(* CODESYS project StorageStation_CECCPrg.project

Project tree, tasks and I/O mapping:
  Device : CECC-D, Festo AG & Co. KG, order no. 574415, version 3.5.4.0
    application Application
      libraries: Standard, * (System); Festo_EXCM_3, 3.5.4.24 (Festo AG & Co. KG); Festo_CVE_3, 3.5.2.11 (Festo AG & Co. KG); VisuDialogs, * (System); CAA CiA 405, 3.5.3.0 (CAA Technical Workgroup)
      task MainTask (cyclic, interval t#20ms, priority 20) calls PLC_PRG
      task VISU_TASK (cyclic, interval 100 ms, priority 30) calls VisuElems.Visu_Prg
      program PLC_PRG [LD]
      global variables Globals
      image pool ImagePool
      global variables Store_Vars
      Visu/
        visualisation Storage_Scheme_new
        visualisation Optionen
        visualisation StorageVisu
        visualisation H_Portal
        visualisation Z_Axis
        visualisation generalControls
      Texts/
        text list Glob_TextList
        text list ARR_ZPOS
        text list ARR_XYPOS
        text list ARR_SPEED
        text list ARR_COLORCHOOSE
      PRGS/
        program prg_hlp [ST]
        program prg_connectCMMO [ST]
        program prg_DriveZAxis [ST]
        program prg_GlobalRef [ST]
        program prg_HomeEXCM [SFC]: Init_active
        program prg_RUNT [ST]
        program prg_HomeZAxis [SFC]
        program prg_startup [ST]
      Driver/
        program prg_DRIVER_CMMO [ST]
        program prg_CALL_DRIVES [FBD]
      EXCM/
        function block EXCM_CCON_CCPOS [ST]
        program EXCM_MANUALJOGG [FBD]
        program EXCM_POSCALC [ST]
        function block EXCM_SCON [ST]
        function block EXCM_SPOS [ST]
      global variables EXCM_Variables
      global variables IN_OUT_VARS
      FB/
        function block FB_Joggin [ST]
        function block FB_DriveZAxis [ST]
        function block FB_Store [ST]
        function block FB_Recognize [ST]
        function block FB_CalcRackPos [ST]
        function block FB_StoreSearch [ST]
        function block FB_DriveHPortal [ST]
        function block FB_SetStorePlace [ST]
        function block FB_Unstore [ST]
        function block FB_ClearStorePlace [ST]
    Onboard : CECC 14I/8O, Festo AG & Co. KG, order no. 
      , version 3.4.5.5
        unmapped channels: Onboard Input, Onboard Output
      Digital Inputs
          unmapped channels: Onboard Input
      Digital Outputs
          output qxGrab : BOOL  // Onboard Output.Byte0.Bit4
          unmapped channels: Onboard Output
    CANbus : CANbus, 3S - Smart Software Solutions GmbH, version 3.5.12.0
        settings: Baudrate = 1000 kbit/s
      CANopen_Manager : CANopen_Manager, 3S - Smart Software Solutions GmbH, version 3.5.10.0
          settings: Sync CycleTime in Microseconds = 8000; Synchronous Window Length = 0; Enable Heartbeat generation = FALSE; ConfigVersion = 50659584
        EXCM_2ST_C3_1 : EXCM-2ST-C3-1, Festo AG & Co. KG, order no. EXCM-CO, version Revision=16#00010000, FileVersion=2.1
            settings: NODEIDSAVED = 1; SDO Timeout = 1000000; EXPERTSETTINGS = TRUE; PDO 16#1400.COBID = 16#0201; PDO 16#1800.COBID = 16#0181; CCON_CPOS.Subindex = 16#00; REC_NR/VELOCITY.Subindex = 16#00; TARGET_POSX.Subindex = 16#00; TARGET_POSY.Subindex = 16#00; SCON_SPOS.Subindex = 16#00; ERROR_NR.Subindex = 16#00; ACT_POSX.Subindex = 16#00; ACT_POSY.Subindex = 16#00; SDO List.Set Guardtime.Index = 16#100C; SDO List.Set Guardtime.Subindex = 16#00; SDO List.Set Guardtime.Value = 16#00000000; SDO List.Set Guardtime.Size = 16; SDO List.Set Guardtime.AbortIfError = FALSE; SDO List.Set Guardtime.JumpToLine = FALSE; SDO List.Set Guardtime.Line = 0; SDO List.Set Lifetime.Index = 16#100D; SDO List.Set Lifetime.Subindex = 16#00; SDO List.Set Lifetime.Value = 16#00000000; SDO List.Set Lifetime.Size = 8; SDO List.Set Lifetime.AbortIfError = FALSE; SDO List.Set Lifetime.JumpToLine = FALSE; SDO List.Set Lifetime.Line = 0; SDO List.Disable Emcy CobID.Index = 16#1014; SDO List.Disable Emcy CobID.Subindex = 16#00; SDO List.Disable Emcy CobID.Value = 16#80000081; SDO List.Disable Emcy CobID.Size = 32; SDO List.Disable Emcy CobID.AbortIfError = FALSE; SDO List.Disable Emcy CobID.JumpToLine = FALSE; SDO List.Disable Emcy CobID.Line = 0; SDO List.Set Emcy CobID.Index = 16#1014; SDO List.Set Emcy CobID.Subindex = 16#00; SDO List.Set Emcy CobID.Value = 16#00000081; SDO List.Set Emcy CobID.Size = 32; SDO List.Set Emcy CobID.AbortIfError = FALSE; SDO List.Set Emcy CobID.JumpToLine = FALSE;
              SDO List.Set Emcy CobID.Line = 0; SDO List.Disable PDO.Index = 16#1400; SDO List.Disable PDO.Subindex = 16#01; SDO List.Disable PDO.Value = 16#80000201; SDO List.Disable PDO.Size = 32; SDO List.Disable PDO.AbortIfError = FALSE; SDO List.Disable PDO.JumpToLine = FALSE; SDO List.Disable PDO.Line = 0; SDO List.Set transmission type.Index = 16#1400; SDO List.Set transmission type.Subindex = 16#02; SDO List.Set transmission type.Value = 16#FF; SDO List.Set transmission type.Size = 8; SDO List.Set transmission type.AbortIfError = FALSE; SDO List.Set transmission type.JumpToLine = FALSE; SDO List.Set transmission type.Line = 0; SDO List.Set and enable COB-ID.Index = 16#1400; SDO List.Set and enable COB-ID.Subindex = 16#01; SDO List.Set and enable COB-ID.Value = 16#00000201; SDO List.Set and enable COB-ID.Size = 32; SDO List.Set and enable COB-ID.AbortIfError = FALSE; SDO List.Set and enable COB-ID.JumpToLine = FALSE; SDO List.Set and enable COB-ID.Line = 0; SDO List.Disable PDO.Index = 16#1800; SDO List.Disable PDO.Subindex = 16#01; SDO List.Disable PDO.Value = 16#80000181; SDO List.Disable PDO.Size = 32; SDO List.Disable PDO.AbortIfError = FALSE; SDO List.Disable PDO.JumpToLine = FALSE; SDO List.Disable PDO.Line = 0; SDO List.Set transmission type.Index = 16#1800; SDO List.Set transmission type.Subindex = 16#02; SDO List.Set transmission type.Value = 16#FF; SDO List.Set transmission type.Size = 8; SDO List.Set transmission type.AbortIfError = FALSE; SDO List.Set transmission type.JumpToLine = FALSE; SDO List.Set transmission type.Line = 0; SDO List.Set inhibit time.Index = 16#1800; SDO List.Set inhibit time.Subindex = 16#03; SDO List.Set inhibit time.Value = 16#0000; SDO List.Set inhibit time.Size = 16;
              SDO List.Set inhibit time.AbortIfError = FALSE; SDO List.Set inhibit time.JumpToLine = FALSE; SDO List.Set inhibit time.Line = 0; SDO List.Set event time.Index = 16#1800; SDO List.Set event time.Subindex = 16#05; SDO List.Set event time.Value = 16#0000; SDO List.Set event time.Size = 16; SDO List.Set event time.AbortIfError = FALSE; SDO List.Set event time.JumpToLine = FALSE; SDO List.Set event time.Line = 0; SDO List.Set and enable COB-ID.Index = 16#1800; SDO List.Set and enable COB-ID.Subindex = 16#01; SDO List.Set and enable COB-ID.Value = 16#00000181; SDO List.Set and enable COB-ID.Size = 32; SDO List.Set and enable COB-ID.AbortIfError = FALSE; SDO List.Set and enable COB-ID.JumpToLine = FALSE; SDO List.Set and enable COB-ID.Line = 0; ConfigVersion = 50659584
            output wEXCM_OUT_CCONCPOS : UINT  // CCON_CPOS
            output wEXCM_OUT_Velocity : UINT  // REC_NR/VELOCITY
            output wEXCM_TargPosX : INT  // TARGET_POSX
            output wEXCM_TargPosY : INT  // TARGET_POSY
            input  wEXCM_IN_SCONSPOS : UINT  // SCON_SPOS
            input  wEXCM_IN_POSX : INT  // ACT_POSX
            input  wEXCM_IN_POSY : INT  // ACT_POSY
            unmapped channels: ERROR_NR
  libraries: VisuSymbols, 3.5.10.0 (System)
  text list GlobalTextList
  5ce3da45-db07-42e7-a21c-a00fff4ed8f6|C:\Users\caha\Pictures\caha.bmp
  data type StorePlace
*)

// StorePlace
TYPE StorePlace :
STRUCT
xUsed: BOOL; //Belegt?
aXVisability: ARRAY[0..3] OF BOOL;	
END_STRUCT
END_TYPE

// Device/Application/Globals
VAR_GLOBAL
	aXvisability: 				ARRAY[0..3] OF BOOL;
	lrZPositionAxis: 			LREAL; 					//Aktuelle Z-Position der Achse		//Current Z position of the axis
	aXTechPositionZ: 			ARRAY[0..2] OF BOOL; 	//Hilfsarray von ZPOS --> Sperrung der Bilder		//ZPOS auxiliary array --> locking of images
	aUSIPositionXY: 			ARRAY[0..3] OF USINT; 	//Listenarray von XYPOS		//List array of XYPOS
	aXVisabilityZPositions:		ARRAY[0..3] OF BOOL;	//3 z positions
	aXVisabilityXYPositions:	ARRAY[1..4] OF BOOL;	//4x positions 
	aXVisabilitySpeedOptions: 	ARRAY[1..3] OF BOOL; 	//Sichtbarkeit Geschwindigkeiten	//Something wrt speed
	usiVisabilityZOptions: 		USINT; 					//Integer für Optionsauswahlt //Option selection 
	usiVisabilitySpeedOptions:	USINT;
	bBitCount: BYTE; //BitCount --> BitCode Input
	
	//MODES
	xModeAuto	:				BOOL;					//Auto - Mode
	xModeIn_Out :				BOOL;					//0 == Store in , 1 == unstore
	xGlobalReset:				BOOL;					// Global Reset.. Reset Fault EXCM Reset Fault CMMO, Reset PRGs
	
	//CMMO DRIVER //Add these drivers for the motor controller
	
	CMMO_DRIVER_1			: CVE.DEV_Driver;
	CMMO_HOME_1				: CVE.DEV_Home;
	CMMO_MOVE_TO_RECORD_1	: CVE.DEV_MoveToRecord;
	CMMO_POWER_1			: CVE.DEV_Power;
	CMMO_READRECORD_1		: CVE.DEV_ReadRecord;
	CMMO_RESET_1			: CVE.DEV_Reset;
	CMMO_SAVE_1				: CVE.DEV_Save;
	CMMO_STOP_1				: CVE.DEV_Stop;
	CMMO_TEACH_1			: CVE.DEV_Teach;
	CMMO_WRITE_RECORD_1		: CVE.DEV_WriteRecord;
	cmmoSTAxis   			: CVE.DEV_AXIS_REF; 	(* axis *)
	CMMO_SW					: CVE.DEV_STATUSWORD;
	cmmoSTReadRecord		: CVE.DEV_RECORD;
											
	xTapForward: 			BOOL;					// Tippen vorwärts	
	xTapBackward: 			BOOL;					// Tippen rückwärts
	xTeach: 				BOOL;					// Teachen
	xReadPositionsOnce: 	BOOL;					// Positionen der Z-Achse aus Motorcontroller lesen
	xConnectCMMO: 			BOOL;					// Z-Achse connectieren
	xBlockConnect: 			BOOL; 					// Verbinden blockieren	
	xDriveZManual: 			BOOL;					// Z-Achse manuell verfahren
	xDrivePositionHPortal: 	BOOL; 					// H-Portal position manuell anfahren
	
	
	FHPP_IN 	AT %IW1: FHPPIN;
	FHPP_OUT 	AT %QW1: FHPPOUT;
	
	EXCM_CAN_DRIVER_1:	 EXCM_CAN_DRIVER;
	EXCM_AXIS: 			 EXCM_AXIS_REF;
	
	usiVisabilityXYOptions: USINT;
	
	bFHPP_IN: 				BYTE;
	bFHPP_OUT: 				BYTE;
	
	xTeachXY: 				BOOL;
	xGlobalReference: 		BOOL; 					// Alles Referenzieren		//Home position defined 
	xStatusGlobalReference:  BOOL;					// Global Referenziert		//At homing position
	xCMMOConnected: 		BOOL;					// CMMO Verbunden 
	xEXCM_HOMED: 			BOOL;					// EXCM Referenziert
	
	xEnAuto: 				BOOL;					// Enable Automatic Mode
	xEinlagern: 			BOOL;					// Einlagern				//Storage mode
	xDriveCMMOFront: 		BOOL;					// CMMO In Position WS 1 fahren
	xDriveCMMORear: 		BOOL;					// Fahre CMMO WS HInten	
	xDriveCMMOGrab: 		BOOL;					// CMMO in Grundstellung (Greifposition fahren)
	
	//What is this?? Not used anywhere!
	xEinlagernComplFB: 		BOOL; 					// Wichtig für Ablauf
	xEinlagerFreigabe: 		BOOL; 					// FREIGABE FÜR AUTOEINLAGERN
	
	xRowPlaceFront: 		BOOL; 					// Lagerplatz vorne oder hinten? TRUE = vorne, FALSE = hinten //Front or rear storage space? TRUE = front, FALSE = rear
	bGlobalRcvData:			BYTE; 					// Empfangenes bzw. erkanntes Werkstück  	//Received or recognized workpiece
	
	//ABLAUF Einalgern
	
	xRackPosReached : 		BOOL; 					
	xGrabPosReached : 		BOOL;
	
	xHomeZAxis: 			BOOL;					// Starte Ablauf zum Referenzieren der Z-Achse		//Start sequence for referencing the Z axis
	
	
	//Positions
	
	xReceiveMode: 			BOOL;					// 0 == selbst erkennen , 1 == Bits Empfangen		//0 == self-detect , 1 == receive bits
	
	
	FB_DriveZAxis1: FB_DriveZAxis;
	FB_DrivePortal_1: FB_DriveHPortal;
	FB_RecognizePart: FB_Recognize;
	FB_StoreSearch1: FB_StoreSearch;
	FB_CalcRackPos1: FB_CalcRackPos;
	FB_Store1: FB_Store;
	
	xClearStore: BOOL;
END_VAR

// Device/Application/Store_Vars
VAR_GLOBAL PERSISTENT RETAIN			//all units are in mm
			 OF StorePlace;
		lrZPositionGrab: 			LREAL := 0.0; 		//Greif-Position							//z Gripping pos
		lrZPositionWorkPieceFront: 	LREAL := 62.96; 		// Position Werkstück vorne				//z Front row position SHOULD'NT THESE BE SAME
		lrZPositionWorkPieceRear: 	LREAL := 116.96; 		// Position Werkstück hinten			//z Rear Row Pos
		

		rXPositionGrab: 			REAL := 591.1;		// Position Werkstück greifen X				//Position Workpiece gripping X
		rYPositionGrab:				REAL := 123.2;		// Position Werkstück greifen Y				// Workpiece position gripping Y
		
		rXPositionWorkPiece1:		REAL := 462.3;		// Position Werkstück1 X					//wORKPIECE1 pOSITION
		rYPositionWorkPiece1:		REAL := 186.2;		// Position Werkstück1 Y	
		
		rXPositionIdle:				REAL :=	448.4;		// Position Werkstück1 X					Idle pos
		rYPositionIdle:				REAL := 123.2;		// Position Werkstück1 Y
		
		rXPositionTransfer:			REAL := 475.9 ;		// Position Übergabe X
		rYPositionTransfer:			REAL := 41.2 ;		// Position Übergabe Y
		
		rPalettenOffset:			REAL := 54;			// Offset auf Palette
		
		//uiDriveSpeed:				UINT := 10;			// Fahrgeschwindigkeit
		//uiGrabSpeed:				UINT := 10;
		//uiLayOnSpeed:				UINT := 5;
		
		aUIColorChoose:		    	ARRAY[0..5] OF UINT;// Fabrauswahl (Dropdown)
		
		// Variablen für CMMO-ST Achse
		lr_GrabPosition: 			LREAL ;			//	Position Greifen
		lr_Workpiece1Position: 		LREAL ;			// 	Position Workpiece 1 Position
		lrStepSize: 				LREAL ;			//  Schrittgröße
		
		rLayOnOffset: 				REAL := 7.5;
		

		cmmoSTRecord			: CVE.DEV_RECORD;
		cmmoSTRecordGrab		: CVE.DEV_RECORD;
		
		cmmoSTRecordFront		: CVE.DEV_RECORD;

		cmmoSTRecordRear		: CVE.DEV_RECORD;
	
		cmmoSTRecordJoggin		: CVE.DEV_RECORD;
END_VAR

// Device/Application/EXCM_Variables
VAR_GLOBAL
	
// ************ CCON _ CPOSS ************
	xEXCM_En_Drive: 				BOOL; 				// Enable Drive
	xEXCM_Stop_Drive: 				BOOL; 				// Stop
	xEXCM_Brake: 					BOOL; 				// Brake on/off
	xEXCM_Axis_Select: 				BOOL; 				// 0 = X-Axis ; 1 = Y-Axis
	xEXCM_Res_Fault: 				BOOL; 				// Reset Fault
	xEXCM_Op_Mode: 					BOOL; 				// 0 = Satzselektion ; 1 = Direktauftraq
	xEXCM_Pos_Mode: 				BOOL; 				// 0 = Positioning Absolute ; 1 Positioning relative
	xEXCM_Start_Task: 				BOOL; 				// Rising Edge = Start Task
	xEXCM_Start_Homing: 			BOOL; 				// Start homing Task
	xEXCM_Jog_Positive: 			BOOL; 				// Jog Positive
	xEXCM_Jog_Negative: 			BOOL; 				// Jog Negative
	
// wEXCM_OUT_CCONCPOS: WORD; 	// Outputword to CANbus
	
	
// ************ SCONSPOS ************	

// wEXCM_IN_SCONSPOS: WORD;		// Inputword CANbus

// ** SCON
	
	xEXCM_STATUS_AckStart: 			BOOL;
	xEXCM_STATUS_MotionComplete: 	BOOL;
	xEXCM_STATUS_InMovement: 		BOOL;
	xEXCM_STATUS_RefPointReached: 	BOOL;

// **SPOS

	xEXCM_STATUS_DriveEnabled: 		BOOL;
	xEXCM_STATUS_Ready: 			BOOL;
	xEXCM_STATUS_Warning: 			BOOL;
	xEXCM_STATUS_Fault: 			BOOL;
	xEXCM_STATUS_VoltagePresent: 	BOOL;
	xEXCM_STATUS_OpMode: 			BOOL;

// ************** OTHERS **************

	rPOSX_Ausgabe: 					REAL;				// Shown Variable Position X
	rPOSY_Ausgabe: 					REAL;				// Shown Variable Position Y
	
	rOutPosX: 						REAL; 
	rOutPosY: 						REAL;

	xManuVisuJogPosY: 				BOOL;
	xManuVisuJogNegY: 				BOOL;
	xManuVisuJogPosX: 				BOOL;
	xManuVisuJogNegX: 				BOOL;
	
	

	
	// ************* Targets ************
	
	rRackPos_X 		 : 				REAL 		:= 0;	// Aktuelle Position zum anfahren
	rRackPos_Y		 : 				REAL 		:= 0;	// ""
	xStorePlaceFound : 				BOOL;
	uiVisuVelocity	 : 				UINT; 				// Geschwindigkeit, manuelles Verfahren
	iTarg_Int_PosX: 				INT;
	iTarg_Int_PosY: 				INT;
	uiSpeed : 						UINT := 200; 		// Geschwindigkeit H-Portal
	uiDriveSpeed :					UINT := 50;
	uiGrabSpeed : 					UINT := 50;
	uiLayOnSpeed : 					UINT := 50;
	xDriveManualXYPos:	 			BOOL;
	xHomeCMMO: 						BOOL;				// Z-Achse Referenzieren
	xCmmoHomed: 					BOOL;				// Z-Achse referenziert
	xHomeExcm: 						BOOL;
	xCMMO_Homed: 					BOOL;				// Z-Achse referenziert#
	xPositionsRead: BOOL;
	xFail: 							BOOL;				// Common Failure
	xPerceived: 					BOOL;				// EMPFANGEN // RECEIVED
	xStartDriveZ: 					BOOL;				// Z_Achse Start_verfahraktion
	uiPositionZToDrive: 			INT;				// Z DrivePosition 0 == Grab; 1 == Position vorne, 2 == Position hinten
	xPositionZReached:				BOOL;				// Z Position erreicht
	xResetZDrive: 					BOOL;				// Reset Z_Verfahraktion
	xGlobalRef: 					BOOL;				// REFERENZIERT
	RS_AUTOL: RS;
	
END_VAR

// Device/Application/IN_OUT_VARS
VAR_GLOBAL
	
	ixReference 		 AT %IX0.0 : BOOL; 					// Referenzieren || Reference
	ixReset 			 AT %IX0.1 : BOOL; 					// Reset Fehler	|| Reset Fail
	ixInOut 			 AT %IX0.2 : BOOL;					// 0 == Einlagern; 1 == Auslagern || 0 == Store; 1 == Unstore
	ixBit0				 AT %IX0.3 : BOOL;					// Bit0 Bitcode
	ixBit1 				 AT %IX0.4 : BOOL;					// Bit1 Bitcode
	ixBit2 				 AT %IX0.5 : BOOL;					// Bit2 Bitcode
	ixStrobe 			 AT %IX0.6 : BOOL; 					// Strobe.. safe Bitcode
	ixMode	    		 AT %IX0.7 : BOOL;					// Auto-/ Manuell Ein-/ Auslagern --> Bei Einlagern: 0 = Erkennt Teil selbst, 1 = BitCode Gibt Lagerfach vor und "Strobe" startet das Lagern || Bei Auslagern --> 0 = Teil wird mit BitCode vorgegeben, 1 = Lagerfach wird mit Bitcode vorgegeben, Strobe startet Auslagervorgang.	
	//Auto/manual Storage/ retrieval --> For storage: 0 = Detects part itself, 1 = BitCode Defines storage compartment and "Strobe" starts storage || For retrieval --> 0 = Part is specified with BitCode, 1 = Storage compartment is specified with Bitcode, Strobe starts retrieval process.	

	qxReferenced 		 AT %QX0.0 : BOOL;
	qxFail				 AT %QX0.1 : BOOL;
	qxStorageBusy		 AT %QX0.2 :BOOL := TRUE ;
	qxStorageFull		 AT %QX0.3 : BOOL;
	
	qxWorkpieceAvailable AT %QX0.5 : BOOL;
	qxPercReflex		 AT %QX0.6 : BOOL;				//Sensors for FB_Recognise, which detects the colour of workpiece and stores in a byte bRcv
	qxPercInduct	 	 AT %QX0.7 : BOOL;

	
	ixStart: BOOL;										// Start Vorgang || Start Action

	
	ixLightGate			 AT %IX1.0		  : BOOL;		// Light-Gate at Recognize Module
	ixPercReflex		 AT %IX1.1		  : BOOL;		// Reflex-Light at Grabposition							
	ixPercInduct		 AT %IX1.2		  : BOOL;		// Inductive Sensor at Recognize Module
	ixWorkpieceAvailable AT %IX1.3	  	  : BOOL;
END_VAR

// Device/Application/PLC_PRG
PROGRAM PLC_PRG// store_vars has the map from real world to here 
//MODES OF Operation
//	xModeAuto	:    				//Auto - Mode
//	xModeIn_Out : 				//0 == Store in , 1 == unstore
//	xGlobalReset:				// Global Reset.. Reset Fault EXCM Reset Fault CMMO, Reset PRGs
//There are 2 modes for controlling the motor controller: Record Selection Mode and Direct Mode
//The bytes for the CPOS and CCON, references on Page 39 of EXCM mnaual

VAR
	Joggin_0: FB_Joggin;
END_VAR
//IF xEXCM_HOMED AND xEXCM_STATUS_RefPointReached THEN

//		xEnAuto := TRUE; //Plc_prg refernce 
//From line 144 from prg_Global REf
//	FB_DrivePortal_1.rPosX := rXPositionIdle ;						//DRIVE TO Idle POSITION
//	FB_DrivePortal_1.rPosY := rYPositionIdle;						//This is algorithm for everymotion 
//	FB_DrivePortal_1.uiEXCM_velocity := uiLayOnSpeed;
//	FB_DrivePortal_1.xStart := TRUE;
//	xEXCM_Start_Task := FB_DrivePortal_1.xStartTask;
//Auto/manual Storage/ retrieval --> For storage: 0 = Detects part itself, 1 = BitCode Defines storage compartment and "Strobe" starts storage || For retrieval --> 0 = Part is specified with BitCode, 1 = Storage compartment is specified with Bitcode, Strobe starts retrieval process

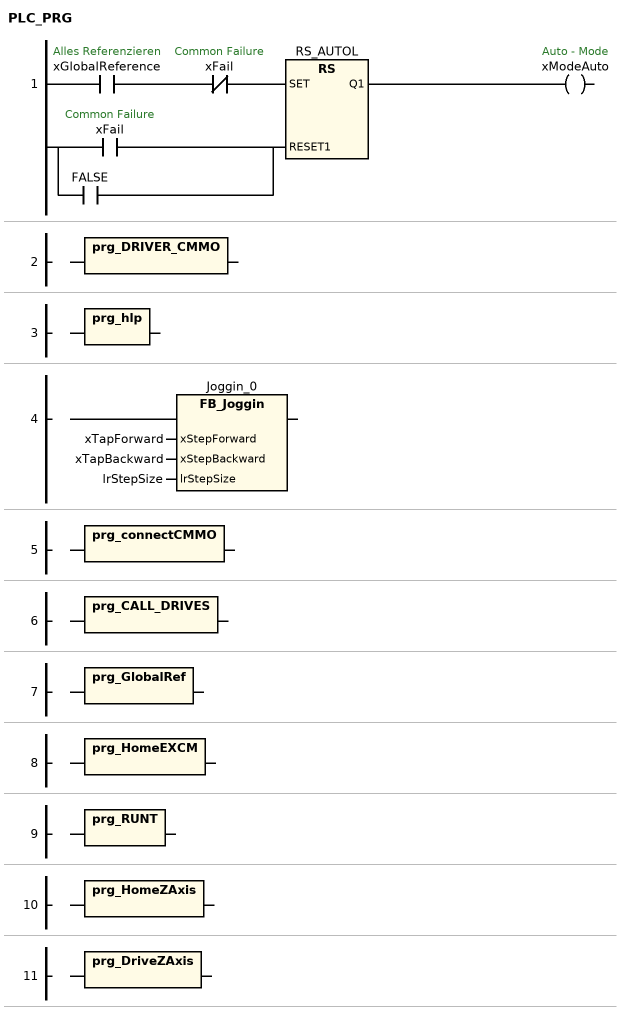
// NETWORK 1
//   xGlobalReference: Alles Referenzieren
//   xFail: Common Failure
//   xModeAuto: Auto - Mode
RS_AUTOL(SET := xGlobalReference AND NOT xFail, RESET1 := xFail OR FALSE); // RS
xModeAuto := RS_AUTOL.Q1;

// NETWORK 2
prg_DRIVER_CMMO();

// NETWORK 3
prg_hlp();

// NETWORK 4
//   xTapForward: Tippen vorwärts
//   xTapBackward: Tippen rückwärts
//   lrStepSize: Schrittgröße
Joggin_0(xStepForward := xTapForward, xStepBackward := xTapBackward, lrStepSize := lrStepSize); // FB_Joggin

// NETWORK 5
prg_connectCMMO();

// NETWORK 6
prg_CALL_DRIVES();

// NETWORK 7
prg_GlobalRef();

// NETWORK 8
prg_HomeEXCM();

// NETWORK 9
prg_RUNT();

// NETWORK 10
prg_HomeZAxis();

// NETWORK 11
prg_DriveZAxis();

END_PROGRAM

// Device/Application/Driver/prg_DRIVER_CMMO
PROGRAM prg_DRIVER_CMMO
//This prg Initialises all the drivers for the CMMO motor controllers
//The drivers are missing right now from this version, they should be named in a fashion of CVE.DEV_<Type>
//The CMMO is controlled in this prg using the CANbus
//CMMO ST Axis??
VAR

	TEST111: LREAL; //LREAL is Floating point number
	//This is just for a test case 
	
END_VAR

CMMO_DRIVER_1(
	xConnect:= , 
	xControl:= , 
	uiPort:= 49700, 
	ipAddr:= '192.168.178.12' , 
	xExternalComCycleEnable:= , 
	xExternalComCycle:= , 
	xIsConnected=> , 
	xHasControl=> , 
	xError=> , 
	eError=> , 
	Axis:= cmmoSTAxis);
	
CMMO_HOME_1(
	xExecute:= , 
	xDone=> , 
	xBusy=> , 
	xError=> , 
	eError=> , 
	Axis:= cmmoSTAxis);
	
CMMO_MOVE_TO_RECORD_1(
	xExecute:= , 
	xDone=> , 
	xBusy=> , 
	xError=> , 
	eError=> , 
	usiRecordNo:= , 
	Axis:= cmmoSTAxis);	

CMMO_POWER_1(
	xEnable:= , 
	xDone=> , 
	xBusy=> , 
	xError=> , 
	eError=> , 
	xEnabled=> , 
	Axis:= cmmoSTAxis);

CMMO_READRECORD_1(
	xExecute:= , 
	xDone=> , 
	xBusy=> , 
	xError=> , 
	eError=> , 
	usiRecordNo:= , 
	Axis:= cmmoSTAxis, 
	Record:= cmmoSTReadRecord);
	
CMMO_RESET_1(
	xExecute:= , 
	xDone=> , 
	xBusy=> , 
	xError=> , 
	eError=> , 
	Axis:= cmmoSTAxis);
	
CMMO_SAVE_1(
	xExecute:= , 
	xDone=> , 
	xBusy=> , 
	xError=> , 
	eError=> , 
	Axis:= cmmoSTAxis);
	
CMMO_STOP_1(
	xExecute:= , 
	xDone=> , 
	xBusy=> , 
	xError=> , 
	eError=> , 
	Axis:= cmmoSTAxis);
	
CMMO_TEACH_1(
	xExecute:= , 
	xDone=> , 
	xBusy=> , 
	xError=> , 
	eError=> , 
	eTarget:= , 
	usiRecordNo:= , 
	Axis:= cmmoSTAxis);
	
CMMO_WRITE_RECORD_1(
	xExecute:= , 
	xDone=> , 
	xBusy=> , 
	xError=> , 
	eError=> , 
	usiRecordNo:= , 
	Axis:= cmmoSTAxis, 
	Record:= cmmoSTRecord);
	
	TEST111 := cmmoSTAxis.lrCurrentPos;
	cmmoSTRecord.eRecordType := 16#10;
	CMMO_SW := CMMOSTAxis.SW;

END_PROGRAM

// Device/Application/PRGS/prg_hlp
PROGRAM prg_hlp
//For the visualisation  
//for the referencing all the taught values
//and driving the robot to the home position 


VAR
	
	uiStep: UINT;
	lr_Workpiece2Position: LREAL;
	uiStep1: UINT;
	uiStep2: UINT;
	uiStep3: UINT;
	i :	INT;
	//FB_DriveManual: FB_Verfahren1;
	
	//FB_DrivePortal: FB_DriveHPortal;
END_VAR

//initialising the sensors 

qxPercInduct 		 := ixPercInduct;
qxPercReflex 		 := ixPercReflex;
qxWorkpieceAvailable := ixWorkpieceAvailable;

(*	FB_DriveManual(
	xStartFahrtFB:= , 
	uiEXCM_velocity:= uiVisuVelocity, 
	rPosX:= , 
	rPosY:= , 
	xMoveComplFB=> );

	
	FB_DrivePortal(
	xStart:= , 
	xReset:= , 
	uiEXCM_Velocity:= , 
	rPosX:= , 
	rPosY:= , 
	xDone=> ,
	xStartTask=> );*)
FB_DrivePortal_1(
	xStart:= , 
	xReset:= , 
	uiEXCM_Velocity:= , 
	rPosX:= , 
	rPosY:= , 
	xDone=> , 
	xStartTask=> );
	
	
FB_DriveZAxis1(uiPosition:= , xStartDrive:= , xReset:= , xPositionReached=> );
		
	
CASE usiVisabilityZOptions OF			//Sichtbarkeit der Positionen in der Visualisierung //There are only 3 options for this 

	1:
	aXVisabilityZPositions[usiVisabilityZOptions] := FALSE;
	aXVisabilityZPositions[2] := TRUE;
	aXVisabilityZPositions[3] := TRUE;
	
	
	2:
	aXVisabilityZPositions[usiVisabilityZOptions] := FALSE;
	aXVisabilityZPositions[1] := TRUE;
	aXVisabilityZPositions[3] := TRUE;
	
	                                                                                                                                                                                                                                                                                                                                                                                                                                                                                                                                                                                                                                                                                                                                                                                                                                                                                                                                                                                                                                                                                                                                                                                                                                                                                                                                                                                                                                                                                                                                                                                                                                                                                                                                                                                                                                                                                                                                                                                                                                                                                                                                                                                                                                                                                                                                                                                                                                                                                                                                                                                                          
	3:	
	aXVisabilityZPositions[usiVisabilityZOptions] := FALSE;
	aXVisabilityZPositions[2] := TRUE;
	aXVisabilityZPositions[1] := TRUE;
	
END_CASE

CASE usiVisabilityXYOptions OF			//Sichtbarkeit der Positionen in der Visualisierung//for the 4 choices of the XY positions from line 253 fro Home, idle , transfer and workpiece
END_CASE

	1:
	aXVisabilityXYPositions[usiVisabilityXYOptions] := FALSE;
	aXVisabilityXYPositions[2] := TRUE;
	aXVisabilityXYPositions[3] := TRUE;
	aXVisabilityXYPositions[4] := TRUE;
	
	2:
	aXVisabilityXYPositions[usiVisabilityXYOptions] := FALSE;
	aXVisabilityXYPositions[1] := TRUE;
	aXVisabilityXYPositions[3] := TRUE;
	aXVisabilityXYPositions[4] := TRUE;
	                                                                                                                                                                                                                                                                                                                                                                                                                                                                                                                                                                                                                                                                                                                                                                                                                                                                                                                                                                                                                                                                                                                                                                                                                                                                                                                                                                                                                                                                                                                                                                                                                                                                                                                                                                                                                                                                                                                                                                                                                                                                                                                                                                                                                                                                                                                                                                                                                                                                                                                                                                                                          
	3:	
	aXVisabilityXYPositions[usiVisabilityXYOptions] := FALSE;
	aXVisabilityXYPositions[2] := TRUE;
	aXVisabilityXYPositions[1] := TRUE;
	aXVisabilityXYPositions[4] := TRUE;
	
	4:
	aXVisabilityXYPositions[usiVisabilityXYOptions] := FALSE;
	aXVisabilityXYPositions[2] := TRUE;
	aXVisabilityXYPositions[1] := TRUE;
	aXVisabilityXYPositions[3] := TRUE;
END_CASE


CASE uiStep OF						 // Positionen in den Speicher des Motorcontrollers schreiben   //Write positions to the motor controller memory initialised in the prg_Driver_CMMO
	0: 
	IF (usiVisabilityZOptions = 1) AND xTeach THEN
		lrZPositionGrab := CMMOSTAxis.lrCurrentPos;
		cmmoSTRecordGrab := CMMOSTRecordJoggin;
		cmmoSTRecord := cmmoSTRecordGrab;
		CMMO_WRITE_RECORD_1.usiRecordNo := 1;
		CMMO_WRITE_RECORD_1.xExecute := TRUE;
		uiStep := 5;
	END_IF
	
	IF (usiVisabilityZOptions = 2) AND xTeach THEN
		lrZPositionWorkPieceFront := CMMOSTAxis.lrCurrentPos;
		cmmoSTRecordFront := CMMOSTRecordJoggin;
		cmmoSTRecord := cmmoSTRecordFront;
		CMMO_WRITE_RECORD_1.usiRecordNo := 2;
		CMMO_WRITE_RECORD_1.xExecute := TRUE;
		uiStep := 5;
	END_IF
	
	IF (usiVisabilityZOptions = 3) AND xTeach THEN
		lrZPositionWorkPieceRear := CMMOSTAxis.lrCurrentPos;
		cmmoSTRecordRear := CMMOSTRecordJoggin;
		cmmoSTRecord := cmmoSTRecordRear;
		CMMO_WRITE_RECORD_1.usiRecordNo := 3;
		CMMO_WRITE_RECORD_1.xExecute := TRUE;
		uiStep := 5;
	END_IF
	
	5:
	CMMO_WRITE_RECORD_1.xExecute := FALSE;
	IF CMMO_WRITE_RECORD_1.xDone AND NOT CMMO_WRITE_RECORD_1.xBusy THEN
		uiStep := 0;
	END_IF
	
END_CASE

CASE uiStep1 OF					// Alle Positionen lesen..
	0:
	IF xReadPositionsOnce THEN
		uiStep1 := 5;
	END_IF

	5:
	CMMO_READRECORD_1.usiRecordNo := 1;
	CMMO_READRECORD_1.xExecute := TRUE;
	uiStep1 := 10;

	10:
	
	CMMO_READRECORD_1.xExecute := FALSE;
	IF CMMO_READRECORD_1.xDone AND NOT CMMO_READRECORD_1.xBusy THEN
		//lrZPositionGrab := CMMOSTReadRecord.lrTarget;
		uiStep1 := 15;
	END_IF

	15: 
	CMMO_READRECORD_1.usiRecordNo := 2;
	CMMO_READRECORD_1.xExecute := TRUE;	
	uiStep1 := 20;

	20:
	CMMO_READRECORD_1.xExecute := FALSE;
	IF CMMO_READRECORD_1.xDone AND NOT CMMO_READRECORD_1.xBusy THEN
		//lrZPositionWorkPieceFront := CMMOSTReadRecord.lrTarget;
		uiStep1 := 25;
	END_IF	
	
	25:
	CMMO_READRECORD_1.usiRecordNo := 3;
	CMMO_READRECORD_1.xExecute := TRUE;
	uiStep1 := 30;
	
	30:
	CMMO_READRECORD_1.xExecute := FALSE;
	IF CMMO_READRECORD_1.xDone AND NOT CMMO_READRECORD_1.xBusy THEN
		//lrZPositionWorkPieceRear := CMMOSTReadRecord.lrTarget;

		uiStep1 := 40;
		
	END_IF
	
	40:
		cmmoSTRecord.eRecordType := 16#10;
		cmmoSTRecord := CMMOSTRecordGrab;
		CMMO_WRITE_RECORD_1.usiRecordNo := 1;
		CMMO_WRITE_RECORD_1.xExecute := TRUE;
		IF CMMO_WRITE_RECORD_1.xDone AND NOT CMMO_WRITE_RECORD_1.xBusy THEN
		CMMO_WRITE_RECORD_1.xExecute := FALSE;
		uiStep1 := 41;
		END_IF
	41:
		cmmoSTRecord := CMMOSTRecordFront;
		CMMO_WRITE_RECORD_1.usiRecordNo := 2;
		CMMO_WRITE_RECORD_1.xExecute := TRUE;
		IF CMMO_WRITE_RECORD_1.xDone AND NOT CMMO_WRITE_RECORD_1.xBusy THEN
		CMMO_WRITE_RECORD_1.xExecute := FALSE;
		uiStep1 := 42;
		END_IF
	42:
		cmmoSTRecord := CMMOSTRecordRear;
		CMMO_WRITE_RECORD_1.usiRecordNo := 3;
		CMMO_WRITE_RECORD_1.xExecute := TRUE;
		IF CMMO_WRITE_RECORD_1.xDone AND NOT CMMO_WRITE_RECORD_1.xBusy THEN
		CMMO_WRITE_RECORD_1.xExecute := FALSE;
		uiStep1 := 45;
		END_IF
		
	45:
		xReadPositionsOnce := FALSE;
		xPositionsRead := TRUE;
		uiStep1 := 0;
END_CASE


CASE uiStep2 OF 	(*DATEN SCHREIBEN*)
		0:
		IF (usiVisabilityZOptions = 1) AND xDriveZManual THEN
			uiStep2 := 5;
		ELSIF (usiVisabilityZOptions = 2) AND xDriveZManual THEN
			uiStep2 := 10;
		ELSIF (usiVisabilityZOptions = 3) AND xDriveZManual THEN
			uiStep2 := 15;
		END_IF
		
		
		5:
		//lrZPositionWorkPieceRear := CMMOSTAxis.lrCurrentPos;
		cmmoSTRecord.eRecordType := 16#10;
		cmmoSTRecord.lrVelocity := 100;
		cmmoSTRecord := CMMOSTRecordGrab;
		CMMO_WRITE_RECORD_1.usiRecordNo := 1;
		CMMO_WRITE_RECORD_1.xExecute := TRUE;
		CMMO_MOVE_TO_RECORD_1.usiRecordNo := 1;
		uiStep2 := 30;
		
		10:
		cmmoSTRecord := CMMOSTRecordFront;
		CMMO_WRITE_RECORD_1.usiRecordNo := 2;
		CMMO_WRITE_RECORD_1.xExecute := TRUE;
		CMMO_MOVE_TO_RECORD_1.usiRecordNo := 2;
		uiStep2 := 30;
		
		15:
		
		cmmoSTRecord := CMMOSTRecordRear;
		CMMO_WRITE_RECORD_1.usiRecordNo := 3;
		CMMO_WRITE_RECORD_1.xExecute := TRUE;
		CMMO_MOVE_TO_RECORD_1.usiRecordNo := 3;
		uiStep2 := 30;
		
		30:
		CMMO_WRITE_RECORD_1.xExecute := FALSE;
		IF CMMO_WRITE_RECORD_1.xDONE AND NOT CMMO_WRITE_RECORD_1.xBusy THEN
			uiStep2  := 35;
		END_IF
		
		35:
		
		CMMO_MOVE_TO_RECORD_1.xExecute := TRUE;
		IF CMMO_MOVE_TO_RECORD_1.xDone AND NOT CMMO_MOVE_TO_RECORD_1.xBusy THEN
			CMMO_MOVE_TO_RECORD_1.xExecute := FALSE;
			xDriveZManual := False;
			uiStep2 := 0;
		END_IF
END_CASE


CASE usiVisabilityXYOptions OF
	
	1:
	IF xTeachXY THEN 
		rXPositionGrab := rPOSX_Ausgabe; //output positions
		rYPositionGrab := rPOSY_Ausgabe;
	END_IF
	
	FB_DrivePortal_1.rPosX := rXPositionGrab;
	FB_DrivePortal_1.rPosY := rYPositionGrab;
	FB_DrivePortal_1.uiEXCM_velocity := uiVisuVelocity;
	FB_DrivePortal_1.xStart := xDriveManualXYPos;
	xEXCM_Start_Task := FB_DrivePortal_1.xStartTask;
		IF FB_DrivePortal_1.xDone THEN
		FB_DrivePortal_1.xStart := FALSE;
		END_IF
	
	2:
	IF xTeachXY THEN
		rXPositionIdle := rPOSX_Ausgabe;
		rYPositionIdle := rPOSY_Ausgabe;
	END_IF
	
	//IF xDriveManualXYPos THEN
	FB_DrivePortal_1.rPosX := rXPositionIdle;
	FB_DrivePortal_1.rPosY := rYPositionIdle;
	FB_DrivePortal_1.uiEXCM_velocity := uiVisuVelocity;
	FB_DrivePortal_1.xStart := xDriveManualXYPos;
	xEXCM_Start_Task := FB_DrivePortal_1.xStartTask;
		IF FB_DrivePortal_1.xDone THEN
		FB_DrivePortal_1.xStart := FALSE;
		END_IF

		
	//END_IF
	
	
	3:
	IF xTeachXY THEN
		rXPositionTransfer := rPOSX_Ausgabe;
		rYPositionTransfer := rPOSY_Ausgabe;
	END_IF

	FB_DrivePortal_1.rPosX := rXPositionTransfer;
	FB_DrivePortal_1.rPosY := rYPositionTransfer;
	FB_DrivePortal_1.uiEXCM_velocity := uiVisuVelocity;
	FB_DrivePortal_1.xStart := xDriveManualXYPos;
	xEXCM_Start_Task := FB_DrivePortal_1.xStartTask;
		IF FB_DrivePortal_1.xDone THEN
		FB_DrivePortal_1.xStart := FALSE;
		END_IF
	4:
	IF xTeachXY THEN
		rXPositionWorkPiece1 := rPOSX_Ausgabe;		
		rYPositionWorkPiece1 := rPOSY_Ausgabe;
	END_IF

	FB_DrivePortal_1.rPosX := rXPositionWorkpiece1;
	FB_DrivePortal_1.rPosY := rYPositionWorkpiece1;
	FB_DrivePortal_1.uiEXCM_velocity := uiVisuVelocity;
	FB_DrivePortal_1.xStart := xDriveManualXYPos;
	xEXCM_Start_Task := FB_DrivePortal_1.xStartTask;
		IF FB_DrivePortal_1.xDone THEN
		FB_DrivePortal_1.xStart := FALSE;
		END_IF
			
END_CASE

IF ixReset THEN
	xGlobalReset := TRUE;
END_IF

CASE uiStep3 OF
	0:
	IF xGlobalReset THEN
		uiStep3 := 5;
	END_IF
	
	5:
	xHomeZAxis := FALSE;
	xStatusGlobalReference := FALSE;
	xGlobalReference := FALSE;

	xEnAuto := FALSE;
	xEXCM_HOMED := FALSE;
	xCMMO_Homed := FALSE;
	FB_RecognizePart.xReset := TRUE;
	xEXCM_En_Drive := FALSE;
	xEXCM_Stop_Drive := FALSE;
	CMMO_DRIVER_1.xControl := FALSE;
	CMMO_DRIVER_1.xConnect :=FALSE;
	CMMO_DRIVER_1.xControl := FALSE;
	CMMO_POWER_1.xEnable := FALSE;
	xCMMOConnected := FALSE;
	xConnectCMMO := FALSE;
	CMMO_DRIVER_1.xConnect := FALSE;
	xBlockConnect := FALSE;
	xHomeCMMO := FALSE;
	xHomeExcm := FALSE;
	uiStep3 := 10;
	
	10:
	
	FB_RecognizePart.xReset := FALSE;
	xGlobalReset := FALSE;
	uiStep3 := 0;
	
END_CASE

bBitCount.0 := ixBit0;
bBitCount.1 := ixBit1;
bBitCount.2 := ixBit2;

END_PROGRAM

// Device/Application/FB/FB_DriveHPortal
FUNCTION_BLOCK FB_DriveHPortal
//for driving the homing portal
VAR_INPUT
	xStart: BOOL;
	xReset: BOOL;
	uiEXCM_Velocity: UINT;
	rPosX : REAL;
	rPosY : REAL;
END_VAR
VAR_OUTPUT
	xDone: BOOL;
	xStartTask: BOOL;
END_VAR
VAR
	rOutPosXCalc: REAL;
	rOutPosYCalc: REAL;
	uiStep: UINT;
	TON_Pulse: TON;
END_VAR

TON_Pulse(IN:= , PT:= T#100MS, Q=> , ET=> );
CASE uiStep OF
	

0:	// Geschwindigkeit von UINT in WORD umwandeln und direkt auf CAN-Adresse schreiben //Convert speed from UINT to WORD and write directly to CAN address
	xDone := FALSE;
	IF xStart THEN
		
	
	wEXCM_OUT_Velocity := UINT_TO_WORD(uiEXCM_velocity);
	
	//Eingangspoisitonen umwandeln und CAN-Adresse schreiben	//Convert input policies and write CAN address
	rOutPosXCalc := rPosX *10;
	rOutPosYCalc := rPosY *10;
	
	iTarg_Int_PosX := REAL_TO_INT(rOutPosXCalc);
	iTarg_Int_PosY := REAL_TO_INT(rOutPosYCalc);
	 
	wEXCM_TargPosX := INT_TO_WORD(iTarg_Int_PosX);
	wEXCM_TargPosY := INT_TO_WORD(iTarg_Int_PosY);
	
	uiStep := 10;
	END_IF

10:
	xStartTask := TRUE;

	TON_Pulse.IN := TRUE;
	IF TON_Pulse.Q THEN
		TON_Pulse.IN := FALSE;
		xStartTask := FALSE;
		
		uiStep := 15;
	END_IF
	
15:
	IF xEXCM_STATUS_MotionComplete AND NOT xEXCM_STATUS_InMovement THEN
		xDone := TRUE;
		TON_Pulse.IN := TRUE;
		IF TON_Pulse.Q THEN
			TON_Pulse.IN := FALSE;
			uiStep := 0;
		END_IF
	END_IF
END_CASE

END_FUNCTION_BLOCK

// Device/Application/FB/FB_Joggin
FUNCTION_BLOCK FB_Joggin
VAR_INPUT
	xStepForward:		BOOL;  			//Step positiv
	xStepBackward:		BOOL;			//Step negativ
	lrStepSize:					LREAL;			//Stepsize
END_VAR
VAR_OUTPUT
	
END_VAR
VAR
	uiStep:				UINT;			// STEP --> CASE
	xForward: BOOL;
	TON_TIMEOUT: TON;
END_VAR

TON_TIMEOUT(IN:= (uiStep=30), PT:= T#4S, Q=> , ET=> );

CASE uiStep OF
	
	0:
	CMMO_RESET_1.xExecute := FALSE;
	CMMOSTRecordJoggin.eRecordType := 16#10;
	CMMOSTRecordJoggin.lrAcceleration := 1;
	CMMOSTRecordJoggin.lrVelocity := 100;
	cmmoSTRecordJoggin.lrTarget := cmmoSTAxis.lrCurrentPos;
		IF xStepForward THEN
			
			xForward := TRUE;
			uiStep := 5;
		ELSIF xStepBackward THEN
			xForward := FALSE;
			uiStep := 5;
		END_IF
	1:
	
	5:
	IF xForward THEN				//Wenn Vorwärts --> Addiere lrStepSize zu der aktuellen Position
		cmmoSTRecordJoggin.lrTarget := cmmoSTAxis.lrCurrentPos + lrStepSize;
		
		IF cmmoSTRecordJoggin.lrTarget > 249 THEN	//Wenn Ergebnis größer 250 --> Alte Position zurückschreiben und Abbruch
			CMMOSTRecordJoggin.lrTarget := 248;	
			uiStep := 50;
		END_IF
	uiStep := 10;
	ELSE						   //Wenn Rückwärts --> Subtrahiere lrStepSize zu der aktuellen Position
		CMMOSTRecordJoggin.lrTarget := cmmoSTAxis.lrCurrentPos - lrStepSize;
		
		IF (CMMOSTRecordJoggin.lrTarget < 0) THEN 	//Wenn Ergebnis kleiner Null --> Alte Position zurückschreiben und Abbruch
			CMMOSTRecordJoggin.lrTarget := 0;	 
			uiStep := 50;
		END_IF
		
	uiStep := 10;
	END_IF
	
	10:
	CMMOSTrecord := CMMOSTRecordJoggin;
	uiStep := 15;
	15:
	CMMO_WRITE_RECORD_1.usiRecordNo := 31;
	CMMO_WRITE_RECORD_1.xExecute := TRUE	;
	uiStep :=20;
	20:
	CMMO_WRite_RECORD_1.xExecute := FALSE;
	IF CMMO_WRITE_RECORD_1.xDONE AND NOT CMMO_WRITE_RECORD_1.xBusy THEN
		uiStep := 25;
	END_IF
	
	25:
	CMMO_MOVE_TO_RECORD_1.usiRecordNo := 31;
	CMMO_MOVE_TO_RECORD_1.xExecute := TRUE;
	uiStep := 30;
	
	30:
		CMMO_MOVE_TO_RECORD_1.xExecute := FALSE;
		IF CMMO_MOVE_TO_RECORD_1.xDone AND NOT CMMO_MOVE_TO_RECORD_1.xBusy THEN
			uiStep := 0;
		END_IF
		xForward := FALSE;
		


		IF TON_TIMEOUT.Q THEN		// TIMEOUT! --> Error Position not reachable
			uiStep := 0;
			CMMO_RESET_1.xExecute := TRUE;
		END_IF
	35:
	
	40:
	
	45:
	
	50:
		//Falls Bereich außerhalb Reichweite
END_CASE

END_FUNCTION_BLOCK

// Device/Application/PRGS/prg_connectCMMO
PROGRAM prg_connectCMMO
//for verifying the connection with the motor driver 
er

VAR
	uiStep: UINT;
	uiStep2: UINT;
END_VAR

IF xGlobalReset THEN
	uiStep := 0;
	uiStep2 := 0;
END_IF

CASE uiStep OF
	0:
	IF xConnectCMMO AND NOT xBlockConnect THEN
		CMMO_DRIVER_1.xConnect := TRUE;
		uiStep := 5;
		xBlockConnect := TRUE;
	END_IF
	
	5:
	IF CMMO_DRIVER_1.xIsConnected THEN
		CMMO_DRIVER_1.xControl := TRUE;
		uiStep:= 10;
	END_IF
	
	10:
	IF CMMO_DRIVER_1.xHasControl THEN
		CMMO_POWER_1.xEnable := TRUE;
		uiStep := 15;
	END_IF
	
	15:
	IF CMMO_POWER_1.xDone AND NOT CMMO_POWER_1.xBusy AND CMMO_POWER_1.xEnabled THEN
		uiStep := 0;
	END_IF
	xCMMOConnected := TRUE;
	
END_CASE

CASE uiStep2 OF
	0:
	IF xHomeCMMO THEN
		CMMO_HOME_1.xExecute := TRUE;
		uiStep2 := 5;
	END_IF
	
	5:
	CMMO_HOME_1.xExecute := FALSE;
	IF CMMO_HOME_1.xDone AND NOT CMMO_HOME_1.xBusy THEN
		uiStep2 := 10;
	END_IF
	
	10:
	xCmmoHomed := TRUE;
	uiStep2 := 0;
	
END_CASE

END_PROGRAM

// Device/Application/Driver/prg_CALL_DRIVES
PROGRAM prg_CALL_DRIVES
VAR
	EXCM_CCON_CCPOS_0: EXCM_CCON_CCPOS;
	EXCM_SPOS_0: EXCM_SPOS;
	EXCM_SCON_0: EXCM_SCON;
	
END_VAR

VAR_INPUT

END_VAR

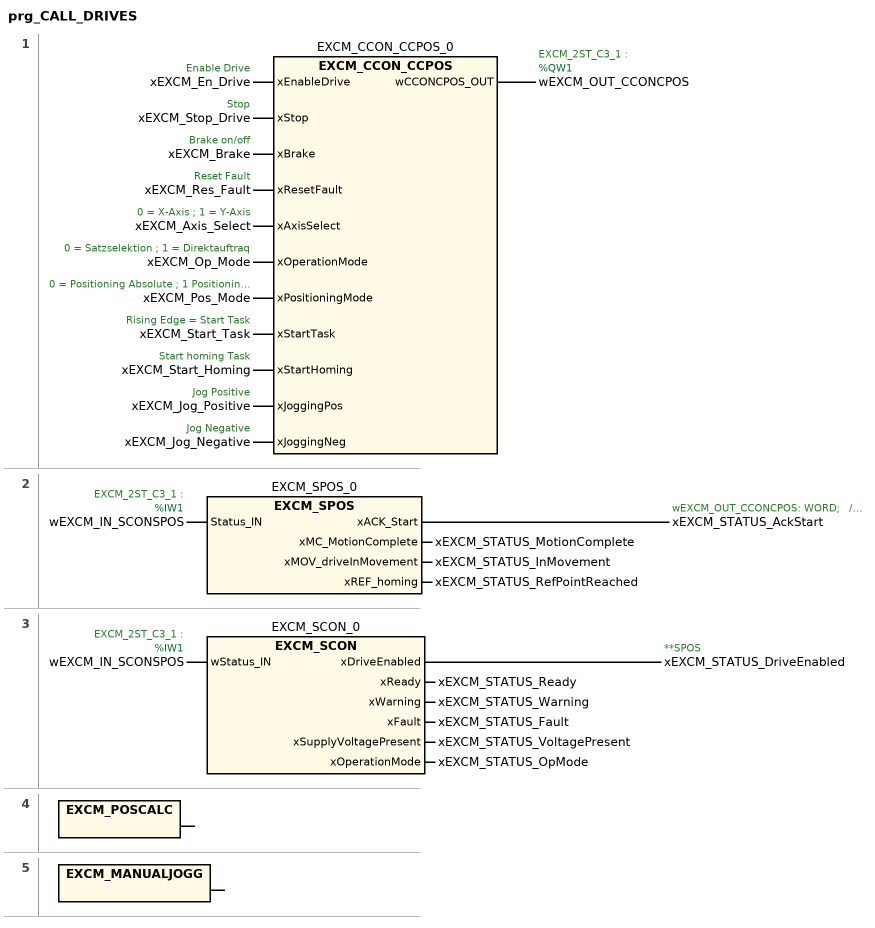
// NETWORK 1
//   xEXCM_En_Drive: Enable Drive
//   xEXCM_Stop_Drive: Stop
//   xEXCM_Brake: Brake on/off
//   xEXCM_Res_Fault: Reset Fault
//   xEXCM_Axis_Select: 0 = X-Axis ; 1 = Y-Axis
//   xEXCM_Op_Mode: 0 = Satzselektion ; 1 = Direktauftraq
//   xEXCM_Pos_Mode: 0 = Positioning Absolute ; 1 Positioning relative
//   xEXCM_Start_Task: Rising Edge = Start Task
//   xEXCM_Start_Homing: Start homing Task
//   xEXCM_Jog_Positive: Jog Positive
//   xEXCM_Jog_Negative: Jog Negative
//   wEXCM_OUT_CCONCPOS: EXCM_2ST_C3_1 : | AT %QW1
EXCM_CCON_CCPOS_0(
    xEnableDrive := xEXCM_En_Drive,
    xStop := xEXCM_Stop_Drive,
    xBrake := xEXCM_Brake,
    xResetFault := xEXCM_Res_Fault,
    xAxisSelect := xEXCM_Axis_Select,
    xOperationMode := xEXCM_Op_Mode,
    xPositioningMode := xEXCM_Pos_Mode,
    xStartTask := xEXCM_Start_Task,
    xStartHoming := xEXCM_Start_Homing,
    xJoggingPos := xEXCM_Jog_Positive,
    xJoggingNeg := xEXCM_Jog_Negative); // EXCM_CCON_CCPOS
wEXCM_OUT_CCONCPOS := EXCM_CCON_CCPOS_0.wCCONCPOS_OUT;

// NETWORK 2
//   wEXCM_IN_SCONSPOS: EXCM_2ST_C3_1 : | AT %IW1
//   xEXCM_STATUS_AckStart: wEXCM_OUT_CCONCPOS: WORD; // Outputword to CANbus ************ SCONSPOS ************ wEXCM_IN_SCONSPOS: WORD; // Inputword CANbus ** SCON
EXCM_SPOS_0(
    Status_IN := wEXCM_IN_SCONSPOS,
    xMC_MotionComplete => xEXCM_STATUS_MotionComplete,
    xMOV_driveInMovement => xEXCM_STATUS_InMovement,
    xREF_homing => xEXCM_STATUS_RefPointReached); // EXCM_SPOS
xEXCM_STATUS_AckStart := EXCM_SPOS_0.xACK_Start;

// NETWORK 3
//   wEXCM_IN_SCONSPOS: EXCM_2ST_C3_1 : | AT %IW1
//   xEXCM_STATUS_DriveEnabled: **SPOS
EXCM_SCON_0(
    wStatus_IN := wEXCM_IN_SCONSPOS,
    xReady => xEXCM_STATUS_Ready,
    xWarning => xEXCM_STATUS_Warning,
    xFault => xEXCM_STATUS_Fault,
    xSupplyVoltagePresent => xEXCM_STATUS_VoltagePresent,
    xOperationMode => xEXCM_STATUS_OpMode); // EXCM_SCON
xEXCM_STATUS_DriveEnabled := EXCM_SCON_0.xDriveEnabled;

// NETWORK 4
EXCM_POSCALC();

// NETWORK 5
EXCM_MANUALJOGG();

END_PROGRAM

// Device/Application/EXCM/EXCM_CCON_CCPOS
FUNCTION_BLOCK EXCM_CCON_CCPOS
VAR_INPUT
xEnableDrive: BOOL;		(* 0 = drive control blocked, 1 = drive control enabled *)
xStop: BOOL;				(* 0 = stop active, 1 = operation enabled *)
xBrake: BOOL;			(* 0 = brake active , 1 = brake released *)
xResetFault: BOOL;		(* Resets error with a rising edge *)	
xAxisSelect: BOOL;		(* 0 = X-Axis , 1 = Y-Axis *)
xOperationMode: BOOL; 	(* 0 = Record Selection , 1 = Direct Mode *)
xPositioningMode: BOOL;	(* 0 = Positioning Absolute, 1 = Positioning relative *)
xStartTask:BOOL; 		(* rising edge: curren setpoint values are accepted and positiong started *)
xStartHoming:BOOL;		(* a rising edge starts homing with the preset parameters *)
xJoggingPos:BOOL	;		(* As long as the bit is set, the drive travels with specified speed in the direction of larger actual values of the axis selected in "axisSelect" *)
xJoggingNeg:BOOL;		(* As long as the bit is set, the drive travels with specified speed in the direction of smaller actual values of the axis selected in "axisSelect" *)

END_VAR
VAR_OUTPUT
wCCONCPOS_OUT: WORD; (* Output of CCON / CPOS *)

END_VAR
VAR
bCCON: BYTE; (* CCON Byte *)
bCPOS: BYTE; (* CPOS Byte *)
pAbs1: POINTER TO BYTE;
abIndex: ARRAY [1..2] OF POINTER TO BYTE;
pRaus: POINTER TO WORD;
END_VAR

pRaus := ADR(wCCONCPOS_OUT);

abIndex[1]:=0;
abIndex[2]:=1;

(*CCON	Byte_1*)
pAbs1     := pRaus + abIndex[1];
bCCON.0   := xEnableDrive;
bCCON.1   := xStop;
bCCON.2	  := xBrake;
bCCON.3   := xResetFault;
bCCON.4   := FALSE;
bCCON.5   := xAxisSelect;
bCCON.6   := xOperationMode;
bCCON.7   := FALSE;
pAbs1^    := bCCON;

(*CPOS	Byte_2*)
pAbs1     := pRaus + abIndex[2];
bCPOS.0   := xPositioningMode;
bCPOS.1   := xStartTask;
bCPOS.2   := xStartHoming;
bCPOS.3   := xJoggingPos;
bCPOS.4   := xJoggingNeg;
bCPOS.5   := FALSE;
bCPOS.6   := FALSE;
bCPOS.7   := FALSE;
pAbs1^    := bCPOS;

END_FUNCTION_BLOCK

// Device/Application/EXCM/EXCM_SPOS
FUNCTION_BLOCK EXCM_SPOS
VAR_INPUT
Status_IN: WORD; (* Input of SCON / SPOS *)
END_VAR
VAR_OUTPUT
	// 1 = ready, 0 = ACK Start
	xACK_Start: BOOL;
	// 1 = Motion complete, 0 = Motion active
	xMC_MotionComplete: BOOL; 
	// 0 = speed of axis < limit , 1 = speed of axis > limit
	xMOV_driveInMovement: BOOL; 
	// 0 = reference run necessary, 1 = reference information available
	xREF_homing: BOOL;
	
END_VAR
VAR
	pSconIn: POINTER TO WORD;
	pAbs: POINTER TO BYTE;
	bSPOS: BYTE;

END_VAR

(* In *)
pSconIn := ADR(Status_IN);	// Pointer auf SSCON / SSTAT

(* SCON *)
pAbs 					:= pSconIn + 1;
bSPOS					:= pAbs^;
// - - - - - - assignment
xACK_Start				:= bSPOS.1;
xMC_MotionComplete		:= bSPOS.2;
xMOV_driveInMovement	:= bSPOS.4;
xREF_homing				:= bSPOS.7;

END_FUNCTION_BLOCK

// Device/Application/EXCM/EXCM_SCON
FUNCTION_BLOCK EXCM_SCON
VAR_INPUT
wStatus_IN: WORD; (* Input of SCON / SPOS *)
END_VAR
VAR_OUTPUT
	// 1 = Drive enabled, 0 = Drive disabled
	xDriveEnabled: BOOL;
	// 1 = positioning enabled, 0 = positioning disabled
	xReady: BOOL; 
	// 0 = no warning, 1 = warning
	xWarning: BOOL; 
	// 0 = no fault, 1 = fault
	xFault: BOOL;
	// 1 = 24V on, 0 = 24V off
	xSupplyVoltagePresent: BOOL;
	
	// 0 = Satzselektion ; 1 = Direktauftrag
	xOperationMode: BOOL;
END_VAR
VAR
	pSconIn: POINTER TO WORD;
	pAbs: POINTER TO BYTE;
	bSCON: BYTE;
END_VAR

(* In *)
psconIn := ADR(wStatus_IN);	// Pointer auf SSCON / SSTAT

(* SCON *)
pAbs 					:= pSconIn + 0;
bSCON					:= pAbs^;
// ------
xDriveEnabled			:= bSCON.0;
xReady					:= bSCON.1;
xWarning				:= bSCON.2;
xFault					:= bSCON.3;
xSupplyVoltagePresent	:= bSCON.4;
xOperationMode			:= bSCON.6;

END_FUNCTION_BLOCK

// Device/Application/EXCM/EXCM_POSCALC
PROGRAM EXCM_POSCALC
VAR
	rPOSX: REAL;
	rPOSY: REAL;
END_VAR

rPOSX := WORD_TO_REAL(wEXCM_IN_POSX); 
rPOSY := WORD_TO_REAL(wEXCM_IN_POSY);

rPOSX_Ausgabe := rPOSX/10;
rPOSY_Ausgabe := rPOSY/10;

	rOutPosX :=  rOutPosX * 10;
	rOutPosY :=  rOutPosY * 10;
	
IF xManuVisuJogPosY THEN 
	xExcm_Axis_Select := TRUE;
END_IF

IF xManuVisuJogNegY THEN
	xExcm_Axis_Select := TRUE;
END_IF
	
IF xManuVisuJogPosX THEN
	xExcm_Axis_Select := FALSE;
END_IF

IF xManuVisuJogNegX THEN
	xExcm_Axis_Select := FALSE;
END_IF

END_PROGRAM

// Device/Application/EXCM/EXCM_MANUALJOGG
PROGRAM EXCM_MANUALJOGG
VAR
END_VAR

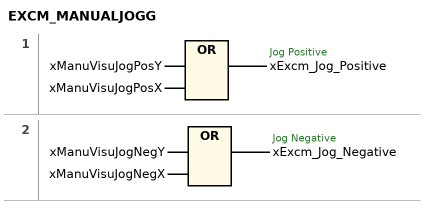
// NETWORK 1
//   xExcm_Jog_Positive: Jog Positive
xExcm_Jog_Positive := xManuVisuJogPosY OR xManuVisuJogPosX;

// NETWORK 2
//   xExcm_Jog_Negative: Jog Negative
xExcm_Jog_Negative := xManuVisuJogNegY OR xManuVisuJogNegX;

END_PROGRAM

// Device/Application/PRGS/prg_GlobalRef
PROGRAM prg_GlobalRef
VAR
	uiStep: UINT;
	uiStep2: UINT;
	xDummy: BOOL;
	TON_Homing: TON;
		TON_WAIT: TON;
	i: INT;
	j: INT;
	k: INT;
	l: INT;
	xFinished: BOOL;
	uiStep3: UINT;
END_VAR

TON_Homing(IN:= , PT:= T#100MS, Q=> , ET=> );
TON_WAIT(IN:= , PT:=T#1000MS , Q=> , ET=> );
qxReferenced := xStatusGlobalReference;

IF xGlobalReset THEN
	uiStep := 0;
	uiStep2:= 0;
	uiStep3:= 0;
	qxFail := FALSE;
END_IF
	
CASE uiStep3 OF


0:
IF xClearStore THEN	
	uiStep3 := 1;
END_IF

//If the storePlace is visible, implies it is filled, after checking all the places
1:
		FOR i:= 0 TO 5 DO
			FOR j:= 0 TO 3 DO
				FOR k:=0 TO 1 DO		
					FOR l:= 0 TO 3 DO
						aStorePlace[i, j, k].aXVisability[l] := TRUE;
					IF i=5 AND j=3 AND k=1 AND l=3 THEN
						xFinished := TRUE;
					EXIT;	
					END_IF
					END_FOR
					aStorePlace[i, j, k].xUsed := FALSE;
											
					
				IF xFinished THEN
					EXIT;
				END_IF
				END_FOR
				IF xFinished THEN
					EXIT;
				END_IF
			END_FOR
			IF xFinished THEN
				EXIT;
			END_IF
		END_FOR

	IF (i=5 AND j=3 AND k = 1 AND l=3) THEN
		uiStep3 := 2;
	END_IF
2:
	xFinished :=FALSE;
	xClearStore := FALSE; 
	uiStep3 := 0;
END_CASE

IF ixReference AND NOT xStatusGlobalReference THEN
	xGlobalReference := TRUE;
END_IF

CASE uiStep OF
	0:	
	IF xGlobalReference THEN
			xConnectCMMO := TRUE;
		IF xCMMOConnected THEN
			xConnectCMMO := FALSE;
			xReadPositionsOnce := TRUE;
			uiStep := 3;
		END_IF
	END_IF
	
	3:
	IF xPositionsRead THEN
	xHomeZAxis := TRUE;
	uiStep := 4;
	END_IF
	
	4:
		cmmoSTRecordGrab.lrTarget := lrZPositionGrab;
		
		// Vorbelegung Speed and Acc Z-Axis
		cmmoSTRecordGrab.lrVelocity := 100;
		cmmoSTRecordGrab.lrAcceleration := 1;
		//
		cmmoSTRecordFront.lrAcceleration := 1;
		cmmoSTRecordFront.lrVelocity := 100;
		//
		cmmoSTRecordRear.lrAcceleration := 1;
		cmmoSTRecordRear.lrVelocity := 100;
		
		cmmoSTRecord := cmmoSTRecordGrab;
		CMMO_WRITE_RECORD_1.usiRecordNo := 1;
		CMMO_WRITE_RECORD_1.xExecute := TRUE;
		uiStep := 5;
	5:
		CMMO_WRITE_RECORD_1.xExecute := FALSE;
		IF CMMO_WRITE_RECORD_1.xDone AND NOT CMMO_WRITE_RECORD_1.xBusy THEN
			uiStep := 6;
		END_IF
	6:
		cmmoSTRecordFront.lrTarget := lrZPositionWorkpieceFront;
		cmmoSTRecord := cmmoSTRecordFront;
		
		CMMO_WRITE_RECORD_1.usiRecordNo := 2;
		CMMO_WRITE_RECORD_1.xExecute := TRUE;
		uiStep := 7;
	7:
		CMMO_WRITE_RECORD_1.xExecute := FALSE;
		IF CMMO_WRITE_RECORD_1.xDone AND NOT CMMO_WRITE_RECORD_1.xBusy THEN
			uiStep := 8;
		END_IF
	8:
		cmmoSTRecordRear.lrTarget := lrZPositionWorkpieceRear;
		cmmoSTRecord := cmmoSTRecordRear;
		CMMO_WRITE_RECORD_1.usiRecordNo := 3;
		CMMO_WRITE_RECORD_1.xExecute := TRUE;
		uiStep := 9;
	9:
	CMMO_WRITE_RECORD_1.xExecute := FALSE;
		IF CMMO_WRITE_RECORD_1.xDone AND NOT CMMO_WRITE_RECORD_1.xBusy THEN
			uiStep := 10;
		END_IF
	

	10:
	xHomeZAxis := FALSE;
	
	IF xCmmoHomed THEN
		xHomeExcm:= TRUE;
		TON_Homing.IN := TRUE;
		IF TON_Homing.Q THEN
		uiStep2 := 5;
		uiStep := 11;	
		END_IF
			
	END_IF
	
	11: 
	TON_HOMING.IN := FALSE;
	xHomeExcm := FALSE;
	qXGrab := TRUE;	
	IF xEXCM_HOMED AND xEXCM_STATUS_RefPointReached THEN

		xEnAuto := TRUE; //Plc_prg refernce 
		uiStep := 12;
	END_IF
	
	12:
	
	IF xFail THEN
		uiStep := 0;
	END_IF

	IF NOT xStatusGlobalReference THEN
	FB_DrivePortal_1.rPosX := rXPositionIdle ;						//DRIVE TO Idle POSITION
	FB_DrivePortal_1.rPosY := rYPositionIdle;						//This is algorithm for everymotion 
	FB_DrivePortal_1.uiEXCM_velocity := uiLayOnSpeed;
	FB_DrivePortal_1.xStart := TRUE;
	xEXCM_Start_Task := FB_DrivePortal_1.xStartTask;
	
	TON_WAIT.IN := TRUE;
	IF FB_DrivePortal_1.xDone AND TON_WAIT.Q THEN
		TON_WAIT.IN := FALSE;
		FB_DrivePortal_1.xStart := FALSE;	
	END_IF
	END_IF
	
	xStatusGlobalReference := TRUE;
	xGlobalReference := FALSE;

		
END_CASE

CASE uiStep2 OF
	0:
	xDummy := TRUE;
	
	5:
	
END_CASE


(*
CASE uiStep2 OF
	
0:
IF ixReference OR xGlobalReference THEN

END_IF

END_CASE*)

END_PROGRAM

// Device/Application/PRGS/prg_HomeEXCM
PROGRAM prg_HomeEXCM
VAR
END_VAR

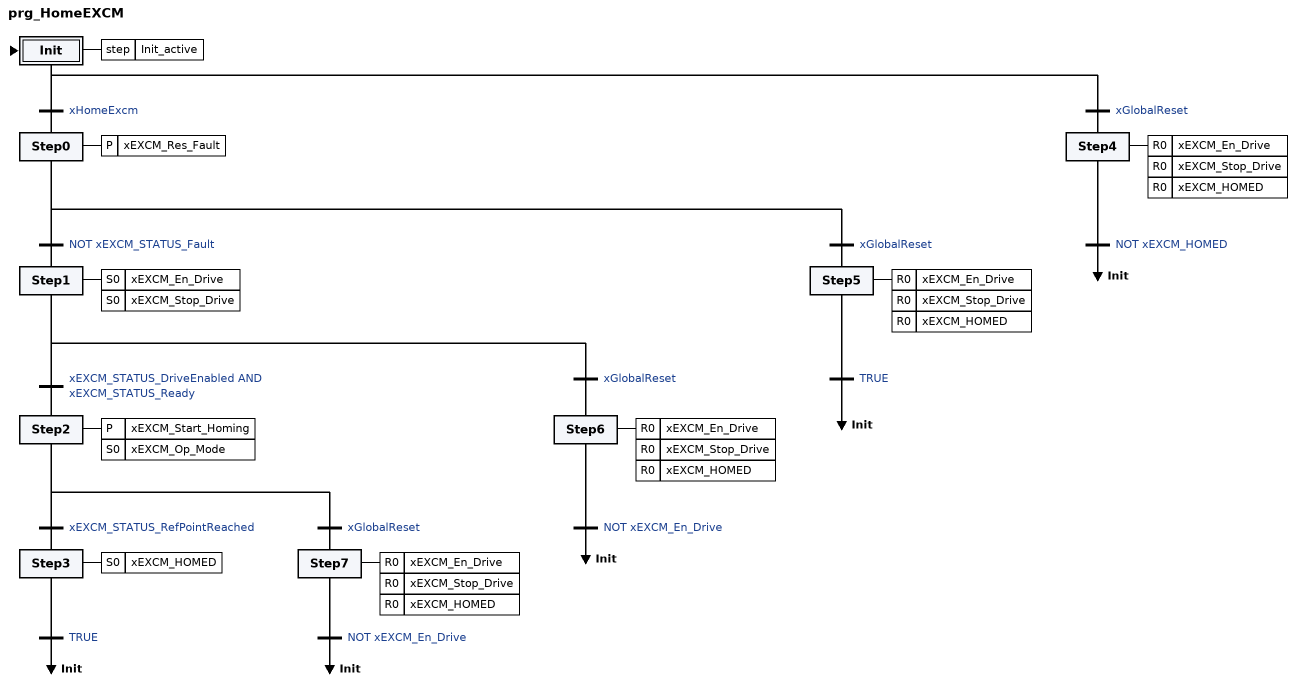
INITIAL_STEP Init:
    Init_active(N);  // step action
END_STEP
TRANSITION FROM Init TO Step0
    := xHomeExcm;
END_TRANSITION
TRANSITION FROM Init TO Step4
    := xGlobalReset;
END_TRANSITION
STEP Step4:
    xEXCM_En_Drive(R0);
    xEXCM_Stop_Drive(R0);
    xEXCM_HOMED(R0);
END_STEP
TRANSITION FROM Step4 TO Init
    := NOT xEXCM_HOMED;
END_TRANSITION
STEP Step0:
    xEXCM_Res_Fault(P);
END_STEP
TRANSITION FROM Step0 TO Step1
    := NOT xEXCM_STATUS_Fault;
END_TRANSITION
TRANSITION FROM Step0 TO Step5
    := xGlobalReset;
END_TRANSITION
STEP Step5:
    xEXCM_En_Drive(R0);
    xEXCM_Stop_Drive(R0);
    xEXCM_HOMED(R0);
END_STEP
TRANSITION FROM Step5 TO Init
    := TRUE;
END_TRANSITION
STEP Step1:
    xEXCM_En_Drive(S0);
    xEXCM_Stop_Drive(S0);
END_STEP
TRANSITION FROM Step1 TO Step2
    := xEXCM_STATUS_DriveEnabled AND xEXCM_STATUS_Ready;
END_TRANSITION
TRANSITION FROM Step1 TO Step6
    := xGlobalReset;
END_TRANSITION
STEP Step6:
    xEXCM_En_Drive(R0);
    xEXCM_Stop_Drive(R0);
    xEXCM_HOMED(R0);
END_STEP
TRANSITION FROM Step6 TO Init
    := NOT xEXCM_En_Drive;
END_TRANSITION
STEP Step2:
    xEXCM_Start_Homing(P);
    xEXCM_Op_Mode(S0);
END_STEP
TRANSITION FROM Step2 TO Step3
    := xEXCM_STATUS_RefPointReached;
END_TRANSITION
TRANSITION FROM Step2 TO Step7
    := xGlobalReset;
END_TRANSITION
STEP Step7:
    xEXCM_En_Drive(R0);
    xEXCM_Stop_Drive(R0);
    xEXCM_HOMED(R0);
END_STEP
TRANSITION FROM Step7 TO Init
    := NOT xEXCM_En_Drive;
END_TRANSITION
STEP Step3:
    xEXCM_HOMED(S0);
END_STEP
TRANSITION FROM Step3 TO Init
    := TRUE;
END_TRANSITION

ACTION Init_active:

END_ACTION

END_PROGRAM

// Device/Application/PRGS/prg_RUNT
PROGRAM prg_RUNT

//First this recognizes the colour and stores it in bGlobalRcvData
//This runs the Storesearch and gets the shelf, row and row place
//then the rack pos is calculated and the place is set visisble in the visualisation and then this is stored in the FB_Store 
//FB_store has 2 programs DriveHPortal and DriveZAxis which use the calculated locations and move the robot

VAR
//	Einlagern: FB_Einlagern; 		// Einlagern FB -> 
	xDummy: BOOL;
	uiStep: UINT;
	R_TRIG_Mode: R_TRIG;
	F_TRIG_Mode: F_TRIG;
	
	xSVMode: BOOL;				//Speichervariable für MODE ..-> Nur geschrieben in STEP 0 oder 5
	xSVInOut: BOOL; 			//Speichervariable für In Out ..-> Nur Abgefragt in STEP 0 oder 5
//	RS_HelpTransparent: 		RS;				// Hilfs RS--> Siehe Programmablauf



	FB_SetStorePlace_1: FB_SetStorePlace;
	
	FB_Unstore1: FB_Unstore;
	FB_ClearStorePlace_1: FB_ClearStorePlace;
	TON_Timeout: TON;
END_VAR

R_TRIG_Mode(CLK:= ixMode, Q=> );
F_TRIG_Mode(CLK:= ixMode, Q=> );

TON_Timeout(IN:= , PT:= , Q=> , ET=> );

IF R_Trig_Mode.Q OR F_TRIG_Mode.Q THEN
		uiStep := 0;
END_IF

IF xGlobalReset THEN
	FB_Store1.xStart := FALSE;
	uiStep := 0;
END_IF

IF FB_StoreSearch1.xErrorStorage THEN
	uiStep := 999;
	ixStart := FALSE;
	// qxFail := TRUE;
END_IF

IF NOT FB_Storesearch1.xErrorStorage AND NOT ixWorkpieceAvailable THEN

//	uiStep := 0;
ixStart := TRUE;			
END_IF



IF xFail OR xGlobalReset OR xEXCM_STATUS_Fault OR CMMO_DRIVER_1.xError THEN
	//xGlobalReference := FALSE;
	//qxFail := TRUE;
	uiStep := 0;
END_IF

FB_CalcRackPos1(
	uiShelf:= , 
	uiRow:= , 
	rPalettOffset:= , 
	rShelfOffset:= , 
	rCalcRackPos_X=> , 
	rCalcRackPos_Y=> );

FB_Unstore1(xStart:= , bRvdData:= , xReset:= , xDone=> );
	
	
FB_StoreSearch1(
	bRcvData:= , 
	xStart:= , 
	xReset:= , 
	uiSearchMode:= , 
	uiStoreMode:= , 
	xStoragePlaceSpotted=> , 
	uiOutShelfNumber=> , 
	uiOutRow=> ,
	uiOutRowPlace=>
	);

FB_SetStorePlace_1(
	uiShelfNumber:= , 
	uiRow:= , 
	uiRowPlace:= , 
	bRcvWorkpiece:= , 
	xSetPlace:= , 
	xReset:= );
	
FB_ClearStorePlace_1(
	uiShelfNumber:= , 
	uiRow:= , 
	uiRowPlace:= , 
	xClearPlace:= , 
	xReset:= );	
	
FB_RecognizePart(xStartRec:=, xReset:= , bWorkpiece=> , xSet=> );	
FB_Store1(xStart:= , bRvdData:= , xReset:= , xDone=> );				
			
FB_CalcRackPos1.rPalettOffset := 54;
FB_CalcRackPos1.rShelfOffset := 90;

IF xEnAuto THEN
	ixStart := TRUE;
	ELSE
	ixStart := FALSE;
END_IF

IF uiStep = 0 OR uiStep = 5 THEN
	xSVMode := ixMode;			//DOUBT with the ixMode
	xSVInOut := ixInOut;		//What store mode store or unstore
END_IF


IF xEnAuto AND xStatusGlobalReference THEN									// Wenn Automatikmodus || If mode automatic  ///////////////////////////////////// NOCH ABÄNDERN VGL. LAGERN BRASIL --> prg_perceive Line 51
// *********************************************************************************************************************************************	
// ******************************************************** EINLAGERN / STORE ******************************************************************
// *********************************************************************************************************************************************
	IF NOT xSVInOut THEN 						// Lagereinstellung 0 == Einlagern, 1 == Auslagern  || Store Setup 0 == store, 1 == unstore
		CASE uiStep OF
			0:
				FB_StoreSearch1.xReset := FALSE;
					FB_RecognizePart.xReset := FALSE;
					
				qxStorageBusy := TRUE;				// Lager beschäftigt setzen || Set Storage busy
				IF ixStart THEN						// Start 
					uiStep := 5;
					bGlobalRcvData := 0;			//The workpiece has entered This var is a BYTE
				END_IF
				FB_SetStorePlace_1.xReset := TRUE;
				
			
				
			5:		
				FB_SetStorePlace_1.xReset := FALSE;
				qxStorageBusy := FALSE;			   // Lager kann Teil empfangen || Storage can receive part-Data
				
				IF NOT xSVMode THEN		   // Wenn selbst erkannt werden soll || Recognition of Workpiece by Station 
					FB_RecognizePart.xStartRec := TRUE;
					IF FB_RecognizePart.xSet THEN
						qxStorageBusy := TRUE;
						bGlobalRcvData := FB_RecognizePart.bWorkpiece;			//bWorkpiece has a value 0,1,2,3 which represents the colour and is stored in bGlobalRcvData
						
						uiStep := 100;
					END_IF
				END_IF
				
				IF xSVMode THEN 			  // Wenn Bitkombination eingegeben wird und mit ixStrobe bestätigt || If Bit combination is set, it will be acknowledged by ixStrobe
						IF ixStrobe AND ixWorkpieceAvailable THEN
						bGlobalRcvData.0 := ixBit0;
						bGlobalRcvData.1 := ixBit1;
						bGlobalRcvData.2 := ixBit2;
						qxStorageBusy := TRUE;
						FB_StoreSearch1.xReset := TRUE;
						uiStep := 200; //wieder auf 200 umstellen
						
					END_IF
				END_IF
			FB_SetStorePlace_1.xReset := FALSE;			//Place reset is set as false
			100:	
		
				
				FB_RecognizePart.xStartRec := FALSE;
				FB_RecognizePart.xReset := TRUE;	
				FB_StoreSearch1.xReset := FALSE;
				uiStep := 101;
							
			101:
				TON_Timeout.PT := T#3S;
				TON_Timeout.IN := (NOT ixWorkpieceAvailable);
				IF TON_Timeout.Q THEN
					FB_RecognizePart.xReset := FALSE;
					uiStep := 0;
				END_IF
				IF ixWorkpieceAvailable THEN
					uiStep := 102;
				END_IF
				
			102:
				//EINSTELLUNGEN SUCHE || SETTINGS SEARCH
				FB_StoreSearch1.uiSearchMode := 0;
				FB_StoreSearch1.uiStoreMode := 0;
				FB_StoreSearch1.bRcvData := bGlobalRcvData;
				FB_StoreSearch1.xStart := TRUE;
				uiStep := 103;
			103:	
				
				// Wenn Platz gefunden... || IF StorePlace found
				IF FB_StoreSearch1.xStoragePlaceSpotted THEN
				FB_CalcRackPos1.uiRow := FB_StoreSearch1.uiOutRow;
				FB_CalcRackPos1.uiShelf := FB_StoreSearch1.uiOutShelfNumber;
				
						
				IF NOT ixMode THEN
					FB_SetStorePlace_1.bRcvWorkpiece := bGlobalRcvData;
				ELSE
					FB_SetStorePlace_1.bRcvWorkpiece := UINT_TO_BYTE(aUIColorChoose[FB_StoreSearch1.uiOutShelfNumber]);
				END_IF;
				FB_SetStorePlace_1.uiShelfNumber := FB_StoreSearch1.uiOutShelfNumber;
				FB_SetStorePlace_1.uiRow := FB_StoreSearch1.uiOutRow;
				FB_SetStorePlace_1.uiRowPlace := FB_StoreSearch1.uiOutRowPlace; 
				
			
				uiStep := 105;
				END_IF
				
				IF FB_StoreSearch1.xErrorStorage THEN
					uiStep := 999;
				END_IF
			105:
				FB_SetStorePlace_1.xSetPlace := TRUE;
				
				FB_RecognizePart.xReset := FALSE;
			//	FB_CalcRackPos1.uiRow := FB_StoreSearch1.uiOutRow;
			//	FB_CalcRackPos1.uiShelf := FB_StoreSearch1.uiOutShelfNumber;
				uiStep := 110;
				
			110:
				FB_SetStorePlace_1.xSetPlace := FALSE;
				FB_StoreSearch1.xStart := FALSE;
				rRackPos_X := FB_CalcRackPos1.rCalcRackPos_X;
				rRackPos_Y := FB_CalcRackPos1.rCalcRackPos_Y;
				uiStep := 115;
			
			115:
				FB_StoreSearch1.xReset := TRUE;
				FB_Store1.xReset := TRUE;
				uiStep := 120;
			
			120:
				FB_StoreSearch1.xReset := FALSE;
				FB_Store1.xReset := FALSE;
				FB_Store1.bRvdData := bGlobalRcvData;
				FB_Store1.xStart := TRUE;
				uiStep := 125;
			
			125:
				IF FB_Store1.xDone THEN
					FB_Store1.xStart := FALSE;
					FB_Store1.xReset := TRUE;
					uiStep := 130;
				END_IF
				
			130:
				FB_RecognizePart.xReset := FALSE;
				FB_Store1.xReset := FALSE;
				FB_SetStorePlace_1.uiStep := 5;
				FB_SetStorePlace_1.xReset := TRUE;
				uiStep := 0;
				
			200:
				//EINSTELLUNGEN SUCHE || SETTINGS SEARCH
				FB_StoreSearch1.xReset := FALSE;
				FB_StoreSearch1.uiSearchMode := 1;
				FB_StoreSearch1.uiStoreMode := 0;
				FB_StoreSearch1.bRcvData := bGlobalRcvData;
				FB_StoreSearch1.xStart := TRUE;
				uiStep := 103;
			
			205:
				FB_CalcRackPos1.uiRow := FB_StoreSearch1.uiOutRow;
				FB_CalcRackPos1.uiShelf := FB_StoreSearch1.uiOutShelfNumber;
				uiStep := 210;
				
			210: 
				FB_StoreSearch1.xStart := FALSE;
				rRackPos_X := FB_CalcRackPos1.rCalcRackPos_X;
				rRackPos_Y := FB_CalcRackPos1.rCalcRackPos_Y;
				uiStep := 215;

			215:
				FB_StoreSearch1.xReset := TRUE;
			999:
				qxStorageFull := TRUE;
				IF NOT FB_StoreSearch1.xErrorStorage AND NOT ixWorkpieceAvailable THEN
					FB_StoreSearch1.xStart := FALSE;
					FB_RecognizePart.xStartRec := FALSE;
					FB_StoreSearch1.xReset := TRUE;
					FB_RecognizePart.xReset := TRUE;
					qxStorageFull := FALSE;
				uiStep := 0;
				END_IF	
				
		END_CASE
	END_IF
// *********************************************************************************************************************************************
// **************************************************** ENDE EINLAGERN / END STORE *************************************************************
// *********************************************************************************************************************************************

// ---------------------------------------------------------------------------------------------------------------------------------------------

// *********************************************************************************************************************************************	
// ******************************************************* AUSLAGERN / UNSTORE *****************************************************************
// *********************************************************************************************************************************************
	IF xSVInOut THEN 							// Lagereinstellung 0 == Einlagern, 1 == Auslagern  || Store Setup 0 == store, 1 == unstore
		CASE uiStep OF
			0:
				FB_StoreSearch1.xReset := FALSE;
				FB_RecognizePart.xReset := FALSE;
				qxStorageBusy := TRUE;				// Lager beschäftigt setzen || Set Storage busy
				IF ixStart THEN						// Start 
					uiStep := 5;
				END_IF
				
			5:		
				qxStorageBusy := FALSE;			   // Lager kann Teil empfangen || Storage can receive part-Data
					IF ixStrobe THEN
						bGlobalRcvData.0 := ixBit0;
						bGlobalRcvData.1 := ixBit1;
						bGlobalRcvData.2 := ixBit2;
						qxStorageBusy := TRUE;
						uiStep := 100;
					END_IF
					FB_ClearStorePlace_1.xReset := TRUE;
					
			100:
				//EINSTELLUNGEN SUCHE || SETTINGS SEARCH
				IF NOT xSVMode THEN
				FB_StoreSearch1.uiSearchMode := 0;
				FB_StoreSearch1.uiStoreMode := 1;
				FB_StoreSearch1.bRcvData := bGlobalRcvData;
				ELSIF xSVMode THEN
				FB_StoreSearch1.uiSearchMode := 1;
				FB_StoreSearch1.uiStoreMode := 1;
				FB_StoreSearch1.bRcvData := bGlobalRcvData;
				END_IF
				
				FB_StoreSearch1.xStart := TRUE;
				IF FB_StoreSearch1.xStoragePlaceSpotted THEN
				FB_CalcRackPos1.uiRow := FB_StoreSearch1.uiOutRow;
				FB_CalcRackPos1.uiShelf := FB_StoreSearch1.uiOutShelfNumber;
				FB_ClearStorePlace_1.uiShelfNumber := FB_StoreSearch1.uiOutShelfNumber;
				FB_ClearStorePlace_1.uiRow := FB_StoreSearch1.uiOutRow;
				FB_ClearStorePlace_1.uiRowPlace := FB_StoreSearch1.uiOutRowPlace;
				
				uiStep := 110;
				END_IF
			110:
				FB_ClearStorePlace_1.xClearPlace := TRUE;
				FB_StoreSearch1.xStart := FALSE;
				rRackPos_X := FB_CalcRackPos1.rCalcRackPos_X;
				rRackPos_Y := FB_CalcRackPos1.rCalcRackPos_Y;
				uiStep := 115;
				
			115:
				FB_StoreSearch1.xReset := TRUE;
				FB_Store1.xReset := TRUE;
				uiStep := 120;
			
			120:
				FB_ClearStorePlace_1.xClearPlace := FALSE;
				FB_StoreSearch1.xReset := FALSE;
				FB_Unstore1.xReset := FALSE;
				FB_Unstore1.bRvdData := bGlobalRcvData;
				FB_Unstore1.xStart := TRUE;
				uiStep := 125;
				
			125:
				IF FB_Unstore1.xDone THEN
					FB_Unstore1.xStart := FALSE;
					FB_Unstore1.xReset := TRUE;
					uiStep := 130;
				END_IF	
			130:
				FB_Unstore1.xReset := FALSE;
				uiStep := 0;
			999:
			qxStorageFull := TRUE;
				IF NOT FB_StoreSearch1.xErrorStorage THEN
					FB_StoreSearch1.xStart := FALSE;
					FB_RecognizePart.xStartRec := FALSE;
					FB_StoreSearch1.xReset := TRUE;
					FB_RecognizePart.xReset := TRUE;
					qxStorageFull := FALSE;
				uiStep := 0;
				END_IF	
		END_CASE
	
// *********************************************************************************************************************************************
// *************************************************** ENDE AUSLAGERN / END UNSTORE ************************************************************
// *********************************************************************************************************************************************
END_IF

	IF xEinlagern THEN
		xDummy := FALSE;
	END_IF
END_IF

END_PROGRAM

// Device/Application/FB/FB_Store
FUNCTION_BLOCK FB_Store
//This drives 2 things 
//z axis and then the DriveHPortal for the other XY axes
VAR_INPUT
	xStart: BOOL;
	bRvdData: BYTE;

	xReset: BOOL;
END_VAR
VAR_OUTPUT
xDone: BOOL;
END_VAR
VAR
	//FB_DrivePortal: FB_Verfahren1;
	uiStep: UINT;
	
	TON_WAIT: TON;
END_VAR

TON_WAIT(IN:= , PT:=T#1000MS , Q=> , ET=> );
IF xGlobalRef THEN
	xStart := FALSE;
	uiStep := 0;
END_IF

CASE uiStep OF
	0:
	IF xStart THEN
		uiStep := 5;
	END_IF
	
	5:	// Sicherstellen, dass Z-Achse eingefahren ist || Check if Z-Axis is retracted
	FB_DriveZAxis1.uiPosition := 1;
	FB_DriveZAxis1.xStartDrive := TRUE;
	uiStep := 6;
	6:
	IF FB_DriveZAxis1.xPositionReached THEN
		FB_DriveZAxis1.xStartDrive := FALSE;
		FB_DriveZAxis1.xReset := TRUE;
		uiStep := 10;
	END_IF

	10: 
	
	FB_DriveZAxis1.xReset := FALSE;
	FB_DrivePortal_1.rPosX := rXPositionIdle;						//DRIVE TO IDLE POSITION
	FB_DrivePortal_1.rPosY := rYPositionIdle;
	FB_DrivePortal_1.uiEXCM_velocity := uiDriveSpeed;
	FB_DrivePortal_1.xStart := TRUE;
	xEXCM_Start_Task := FB_DrivePortal_1.xStartTask;
	
	qxGrab := TRUE;
	TON_WAIT.IN := TRUE;
	IF FB_DrivePortal_1.xDone AND TON_WAIT.Q THEN
		TON_WAIT.IN := FALSE;
		FB_DrivePortal_1.xStart := FALSE;
		uiStep := 15;
	END_IF
	
	
	15:
	FB_DriveZAxis1.xReset := FALSE;
	FB_DrivePortal_1.rPosX := rXPositionGrab;						//DRIVE TO GRAB POSITION
	FB_DrivePortal_1.rPosY := rYPositionGrab;
	FB_DrivePortal_1.uiEXCM_velocity := uiDriveSpeed;
	FB_DrivePortal_1.xStart := TRUE;
	xEXCM_Start_Task := FB_DrivePortal_1.xStartTask;
	
	TON_WAIT.IN := TRUE;
		IF FB_DrivePortal_1.xDone AND TON_WAIT.Q THEN
		TON_WAIT.IN := FALSE;
		FB_DrivePortal_1.xStart := FALSE;
		qxGrab := FALSE;
		uiStep := 20;
		END_IF



	
	20: 
	FB_DrivePortal_1.rPosX := rXPositionIdle;						//DRIVE TO IDLE POSITION AGAIN
	FB_DrivePortal_1.rPosY := rYPositionIdle;
	FB_DrivePortal_1.uiEXCM_velocity := uiDriveSpeed;
	FB_DrivePortal_1.xStart := TRUE;
	xEXCM_Start_Task := FB_DrivePortal_1.xStartTask;
	
	TON_WAIT.IN := TRUE;
	IF FB_DrivePortal_1.xDone AND TON_WAIT.Q THEN
		TON_WAIT.IN := FALSE;
		FB_DrivePortal_1.xStart := FALSE;
		uiStep := 25;
	END_IF
	
		
	25:
	FB_DrivePortal_1.rPosX := (rRackPos_X - rLayonOffset);						//DRIVE TO RACK POSITION -(minus) OFFSET
	FB_DrivePortal_1.rPosY := rRackPos_Y;
	FB_DrivePortal_1.uiEXCM_velocity := uiDriveSpeed;
	FB_DrivePortal_1.xStart := TRUE;
	xEXCM_Start_Task := FB_DrivePortal_1.xStartTask;
	
	TON_WAIT.IN := TRUE;
	IF FB_DrivePortal_1.xDone AND TON_WAIT.Q THEN
		TON_WAIT.IN := FALSE;
		FB_DrivePortal_1.xStart := FALSE;
		uiStep := 30;
	END_IF

	30:
	IF NOT xRowPlaceFront THEN
		FB_DriveZAxis1.uiPosition := 2;
	ELSE
		FB_DriveZAxis1.uiPosition := 3;
	END_IF
	uiStep := 35;
	
	
	35:

	
	FB_DriveZAxis1.xStartDrive := TRUE;
	uiStep := 36;
	
	36:
	IF FB_DriveZAxis1.xPositionReached THEN
		FB_DriveZAxis1.xStartDrive := FALSE;
		
		uiStep := 40;
	END_IF

	
	
	40:
	FB_DriveZAxis1.xReset := TRUE;
	//FB_DrivePortal_1.xReset := TRUE;
//	FB_DriveZAxis1.xReset := FALSE;
	FB_DrivePortal_1.rPosX := rRackPos_X ;						//DRIVE TO RACK POSITION
	FB_DrivePortal_1.rPosY := rRackPos_Y;
	FB_DrivePortal_1.uiEXCM_velocity := uiLayOnSpeed;
	FB_DrivePortal_1.xStart := TRUE;
	xEXCM_Start_Task := FB_DrivePortal_1.xStartTask;
	
	TON_WAIT.IN := TRUE;
	IF FB_DrivePortal_1.xDone AND TON_WAIT.Q THEN
		TON_WAIT.IN  := FALSE;
		FB_DrivePortal_1.xStart := FALSE;
		qxGrab := TRUE;
		uiStep := 41;
		FB_DriveZAxis1.xReset := FALSE;
	END_IF
	FB_DriveZAxis1.uiPosition := 1;
	
	41:
	FB_DrivePortal_1.rPosX := (rRackPos_X - rLayonOffset);						//DRIVE TO RACK POSITION -(minus) OFFSET
	FB_DrivePortal_1.rPosY := rRackPos_Y;
	FB_DrivePortal_1.uiEXCM_velocity := uiDriveSpeed;
	FB_DrivePortal_1.xStart := TRUE;
	xEXCM_Start_Task := FB_DrivePortal_1.xStartTask;
	
	TON_WAIT.IN := TRUE;
	IF FB_DrivePortal_1.xDone AND TON_WAIT.Q THEN
		TON_WAIT.IN := FALSE;
		FB_DrivePortal_1.xStart := FALSE;
		uiStep := 42;
	END_IF
	42:
	uiStep := 45;

	45:
	TON_WAIT.IN := FALSE;
	FB_DriveZAxis1.xStartDrive := TRUE;
	uiStep := 46;
	
	46:
	TON_WAIT.IN := TRUE; 
	IF FB_DriveZAxis1.xPositionReached AND TON_WAIT.Q THEN
		TON_WAIT.IN := FALSE;
		FB_DriveZAxis1.xStartDrive := FALSE;
		
		uiStep := 50;
	END_IF
	

	50:
	FB_DriveZAxis1.xReset := TRUE;
	FB_DrivePortal_1.rPosX := rXPositionIdle ;						//DRIVE TO Idle POSITION
	FB_DrivePortal_1.rPosY := rYPositionIdle;
	FB_DrivePortal_1.uiEXCM_velocity := uiDriveSpeed;
	FB_DrivePortal_1.xStart := TRUE;
	xEXCM_Start_Task := FB_DrivePortal_1.xStartTask;
	
	TON_WAIT.IN := TRUE;
	IF FB_DrivePortal_1.xDone AND TON_WAIT.Q THEN
		TON_WAIT.IN := FALSE;
		FB_DrivePortal_1.xStart := FALSE;
		qxGrab := TRUE;
		uiStep := 55;
		FB_DriveZAxis1.xReset := FALSE;
	END_IF
	
	55:
	
	xDone := TRUE;
	
	IF xReset THEN
	xDone := FALSE;
	uiStep := 0;

	END_IF	
	(*	
	IF FB_DrivePortal.xMoveComplFB THEN
		FB_DrivePortal.xStartFahrtFB := FALSE;
		qxGrab := TRUE;										// Greifer öffnen
		uiStep := 55;										// ABSETZEN EINPLANEN, WS in ARRAY zu setzen!
	END_IF
	
	55:
	FB_DrivePortal.rPosX := rXPositionIdle;						//DRIVE TO RACK POSITION
	FB_DrivePortal.rPosY := rYPositionIdle;
	FB_DrivePortal.uiEXCM_velocity := uiLayOnSpeed;
	FB_DrivePortal.xStartFahrtFB := TRUE;
	uiStep := 60;
	
	60:
	IF FB_DrivePortal.xMoveComplFB THEN
		FB_DrivePortal.xStartFahrtFB := FALSE;
		qxGrab := TRUE;			// Greifer öffnen	
		xDone := TRUE;															// ABSETZEN EINPLANEN, WS in ARRAY zu setzen!
	END_IF
	IF xReset AND NOT xStart THEN
		xDone := FALSE;
		uiStep := 0;
	END_IF
*)	
END_CASE

END_FUNCTION_BLOCK

// Device/Application/FB/FB_SetStorePlace
FUNCTION_BLOCK FB_SetStorePlace
VAR_INPUT
	uiShelfNumber:		UINT;
	uiRow:				UINT;
	uiRowPlace:			UINT;
	bRcvWorkpiece:		BYTE;
	xSetPlace:		 	BOOL;
	xReset: 			BOOL;
	uiStep: 			UINT;
END_VAR
VAR_OUTPUT
END_VAR
VAR
	//uiStep: UINT;
	i: BYTE;
	xSetReady: BOOL;
	
END_VAR

CASE uiStep OF
	0:
	IF xSetPlace THEN
		uiStep := 1;
	END_IF
	
	1:
	aStorePlace[uiShelfNumber, uiRow, uiRowPlace].xUsed := TRUE;				//This sets the colour of the workpiece according to the bRcvWorkpiece
	FOR i:=0 TO 3 DO
		IF NOT i = bRcvWorkpiece THEN
			aStorePlace[uiShelfNumber, uiRow, uiRowPlace].aXVisability[i] := TRUE;
			IF i = 3 OR i = 4 THEN
				uiStep := 5;
			END_IF
		ELSIF i = bRcvWorkpiece THEN
			aStorePlace[uiShelfNumber, uiRow, uiRowPlace].aXVisability[i] := FALSE;
			IF i = 3 OR i = 4 THEN
				uiStep := 5;
			END_IF
		END_IF
		
	END_FOR
	
	5:
	IF xReset THEN
		i := 0;
		uiStep := 0;
	END_IF
END_CASE

END_FUNCTION_BLOCK

// Device/Application/FB/FB_Unstore
FUNCTION_BLOCK FB_Unstore
VAR_INPUT
	xStart: BOOL;
	bRvdData: BYTE;
	
	xReset: BOOL;
END_VAR
VAR_OUTPUT
xDone: BOOL;
END_VAR
VAR
	//FB_DrivePortal: FB_Verfahren1;
	uiStep: UINT;
	
	TON_WAIT: TON;
END_VAR

TON_WAIT(IN:= , PT:=T#200MS , Q=> , ET=> );
IF xFail OR xGlobalRef THEN
	xStart := FALSE;
	uiStep := 0;
END_IF

CASE uiStep OF
	0:
	IF xStart THEN
		uiStep := 5;
	END_IF
	
	5:	// Sicherstellen, dass Z-Achse eingefahren ist || Check if Z-Axis is retracted
	FB_DriveZAxis1.uiPosition := 1;
	FB_DriveZAxis1.xStartDrive := TRUE;
	uiStep := 6;
	6:
	IF FB_DriveZAxis1.xPositionReached THEN
		FB_DriveZAxis1.xStartDrive := FALSE;
		FB_DriveZAxis1.xReset := TRUE;
		uiStep := 10;
	END_IF

	10:
	(*
	FB_DriveZAxis1.xReset := FALSE;
	FB_DrivePortal_1.rPosX := rXPositionIdle;						//DRIVE TO IDLE POSITION
	FB_DrivePortal_1.rPosY := rYPositionIdle;
	FB_DrivePortal_1.uiEXCM_velocity := uiDriveSpeed;
	FB_DrivePortal_1.xStart := TRUE;
	xEXCM_Start_Task := FB_DrivePortal_1.xStartTask;
	
	qxGrab := TRUE;
	TON_WAIT.IN := TRUE;
	IF FB_DrivePortal_1.xDone AND TON_WAIT.Q THEN
		TON_WAIT.IN := FALSE;
		FB_DrivePortal_1.xStart := FALSE;*)
		uiStep := 15;
	//END_IF
	
	
	15:










(*	FB_DriveZAxis1.xReset := FALSE;
	FB_DrivePortal_1.rPosX := rXPositionGrab;						//DRIVE TO GRAB POSITION
	FB_DrivePortal_1.rPosY := rYPositionGrab;
	FB_DrivePortal_1.uiEXCM_velocity := uiDriveSpeed;
	FB_DrivePortal_1.xStart := TRUE;
	xEXCM_Start_Task := FB_DrivePortal_1.xStartTask;
	
	TON_WAIT.IN := TRUE;
		IF FB_DrivePortal_1.xDone AND TON_WAIT.Q THEN
		TON_WAIT.IN := FALSE;
		FB_DrivePortal_1.xStart := FALSE;
		qxGrab := FALSE;*)
		uiStep := 20;
		//END_IF



	
	20: 
(*	FB_DrivePortal_1.rPosX := rXPositionIdle;						//DRIVE TO IDLE POSITION AGAIN
	FB_DrivePortal_1.rPosY := rYPositionIdle;
	FB_DrivePortal_1.uiEXCM_velocity := uiDriveSpeed;
	FB_DrivePortal_1.xStart := TRUE;
	xEXCM_Start_Task := FB_DrivePortal_1.xStartTask;
	
	TON_WAIT.IN := TRUE;
	IF FB_DrivePortal_1.xDone AND TON_WAIT.Q THEN
		TON_WAIT.IN := FALSE;
		FB_DrivePortal_1.xStart := FALSE;
		uiStep := 25;
	END_IF
*)	
	uiStep := 25;
		
	25:
	FB_DrivePortal_1.rPosX := rRackPos_X;						//DRIVE TO RACK POSITION
	FB_DrivePortal_1.rPosY := rRackPos_Y;
	FB_DrivePortal_1.uiEXCM_velocity := uiDriveSpeed;
	FB_DrivePortal_1.xStart := TRUE;
	xEXCM_Start_Task := FB_DrivePortal_1.xStartTask;
	
	TON_WAIT.IN := TRUE;
	IF FB_DrivePortal_1.xDone AND TON_WAIT.Q THEN
		TON_WAIT.IN := FALSE;
		FB_DrivePortal_1.xStart := FALSE;
		uiStep := 30;
	END_IF

	30:
	IF NOT xRowPlaceFront THEN
		FB_DriveZAxis1.uiPosition := 2;
	ELSE
		FB_DriveZAxis1.uiPosition := 3;
	END_IF
	uiStep := 35;
	
	
	35:

	
	FB_DriveZAxis1.xStartDrive := TRUE;
	uiStep := 36;
	
	36:
	IF FB_DriveZAxis1.xPositionReached THEN
		FB_DriveZAxis1.xStartDrive := FALSE;
		qxGrab := FALSE;
		uiStep := 40;
	END_IF

	
	
	40:
	FB_DriveZAxis1.xReset := TRUE;
	//FB_DrivePortal_1.xReset := TRUE;
//	FB_DriveZAxis1.xReset := FALSE;
	FB_DrivePortal_1.rPosX := (rRackPos_X-rLayOnOffSet) ;						//DRIVE TO RACK POSITION - OFFSET
	FB_DrivePortal_1.rPosY := rRackPos_Y;
	FB_DrivePortal_1.uiEXCM_velocity := uiLayOnSpeed;
	FB_DrivePortal_1.xStart := TRUE;
	xEXCM_Start_Task := FB_DrivePortal_1.xStartTask;
	
	TON_WAIT.IN := TRUE;
	IF FB_DrivePortal_1.xDone AND TON_WAIT.Q THEN
		TON_WAIT.IN  := FALSE;
		FB_DrivePortal_1.xStart := FALSE;
		//qxGrab := TRUE;
		uiStep := 45;
		FB_DriveZAxis1.xReset := FALSE;
	END_IF
	FB_DriveZAxis1.uiPosition := 1;
	45:
	TON_WAIT.IN := FALSE;
	FB_DriveZAxis1.xStartDrive := TRUE;
	uiStep := 46;
	
	46:
	TON_WAIT.IN := TRUE; 
	IF FB_DriveZAxis1.xPositionReached AND TON_WAIT.Q THEN
		TON_WAIT.IN := FALSE;
		FB_DriveZAxis1.xStartDrive := FALSE;
		
		uiStep := 47;
	END_IF
	
	47:
	FB_DriveZAxis1.xReset := TRUE;
	FB_DrivePortal_1.rPosX := rXPositionTransfer ;						//DRIVE TO Idle POSITION
	FB_DrivePortal_1.rPosY := rYPositionTransfer;
	FB_DrivePortal_1.uiEXCM_velocity := uiDriveSpeed;
	FB_DrivePortal_1.xStart := TRUE;
	xEXCM_Start_Task := FB_DrivePortal_1.xStartTask;
	
	TON_WAIT.IN := TRUE;
	IF FB_DrivePortal_1.xDone AND TON_WAIT.Q THEN
		TON_WAIT.IN := FALSE;
		FB_DrivePortal_1.xStart := FALSE;
		qxGrab := TRUE;
		uiStep := 50;
		FB_DriveZAxis1.xReset := FALSE;
	END_IF
	

	50:
	FB_DriveZAxis1.xReset := TRUE;
	FB_DrivePortal_1.rPosX := rXPositionIdle ;						//DRIVE TO Idle POSITION
	FB_DrivePortal_1.rPosY := rYPositionIdle;
	FB_DrivePortal_1.uiEXCM_velocity := uiDriveSpeed;
	FB_DrivePortal_1.xStart := TRUE;
	xEXCM_Start_Task := FB_DrivePortal_1.xStartTask;
	
	TON_WAIT.IN := TRUE;
	IF FB_DrivePortal_1.xDone AND TON_WAIT.Q THEN
		TON_WAIT.IN := FALSE;
		FB_DrivePortal_1.xStart := FALSE;
		qxGrab := TRUE;
		uiStep := 51;
		FB_DriveZAxis1.xReset := FALSE;
	END_IF
		
	51:
	IF rPOSX_Ausgabe < (rXPositionIdle +1) AND rPOSX_Ausgabe > (rXPositionIdle - 1) AND rPOSY_Ausgabe < (rYPositionIdle +1) AND rPOSY_Ausgabe > (rYPositionIdle -1) THEN
	uistep:=55;
	ELSE
	uistep:=50;
	END_IF
	
	
	55:
	
	xDone := TRUE;
	
	IF xReset THEN
	xDone := FALSE;
	uiStep := 0;
	
	END_IF	
	(*	
	IF FB_DrivePortal.xMoveComplFB THEN
		FB_DrivePortal.xStartFahrtFB := FALSE;
		qxGrab := TRUE;										// Greifer öffnen
		uiStep := 55;										// ABSETZEN EINPLANEN, WS in ARRAY zu setzen!
	END_IF
	
	55:
	FB_DrivePortal.rPosX := rXPositionIdle;						//DRIVE TO RACK POSITION
	FB_DrivePortal.rPosY := rYPositionIdle;
	FB_DrivePortal.uiEXCM_velocity := uiLayOnSpeed;
	FB_DrivePortal.xStartFahrtFB := TRUE;
	uiStep := 60;
	
	60:
	IF FB_DrivePortal.xMoveComplFB THEN
		FB_DrivePortal.xStartFahrtFB := FALSE;
		qxGrab := TRUE;			// Greifer öffnen	
		xDone := TRUE;															// ABSETZEN EINPLANEN, WS in ARRAY zu setzen!
	END_IF
	IF xReset AND NOT xStart THEN
		xDone := FALSE;
		uiStep := 0;
	END_IF
*)	
END_CASE

END_FUNCTION_BLOCK

// Device/Application/FB/FB_ClearStorePlace
FUNCTION_BLOCK FB_ClearStorePlace
VAR_INPUT
	uiShelfNumber: UINT;
	uiRow: UINT;
	uiRowPlace: UINT;
	xClearPlace: BOOL;
	xReset: BOOL;
END_VAR
VAR_OUTPUT
END_VAR
VAR
	uiStep: UINT;
	i: INT;
END_VAR

CASE uiStep OF
	0:
	IF xClearPlace THEN
		uiStep := 1;
	END_IF
	
	1:
	aStorePlace[uiShelfNumber, uiRow, uiRowPlace].xUsed := FALSE;
	FOR i:=0 TO 3 DO
			aStorePlace[uiShelfNumber, uiRow, uiRowPlace].aXVisability[i] := TRUE;
			IF i=3 THEN
				uiStep := 5;
			END_IF
	END_FOR
	
	5:
	IF xReset THEN
		i := 0;
		uiStep := 0;
	END_IF
END_CASE

END_FUNCTION_BLOCK

// Device/Application/PRGS/prg_HomeZAxis
PROGRAM prg_HomeZAxis
VAR
END_VAR

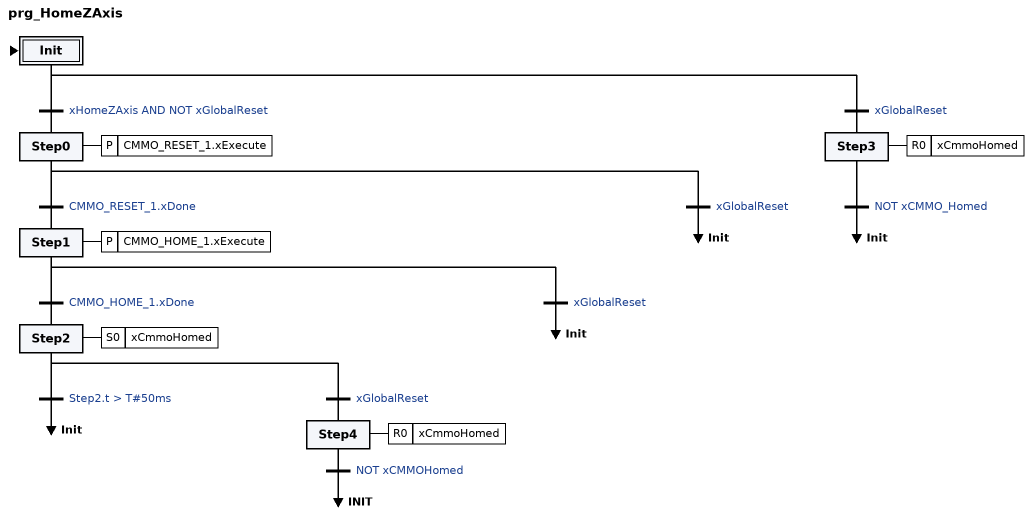
INITIAL_STEP Init:
END_STEP
TRANSITION FROM Init TO Step0
    := xHomeZAxis AND NOT xGlobalReset;
END_TRANSITION
TRANSITION FROM Init TO Step3
    := xGlobalReset;
END_TRANSITION
STEP Step3:
    xCmmoHomed(R0);
END_STEP
TRANSITION FROM Step3 TO Init
    := NOT xCMMO_Homed;
END_TRANSITION
STEP Step0:
    CMMO_RESET_1.xExecute(P);
END_STEP
TRANSITION FROM Step0 TO Step1
    := CMMO_RESET_1.xDone;
END_TRANSITION
TRANSITION FROM Step0 TO Init
    := xGlobalReset;
END_TRANSITION
STEP Step1:
    CMMO_HOME_1.xExecute(P);
END_STEP
TRANSITION FROM Step1 TO Step2
    := CMMO_HOME_1.xDone;
END_TRANSITION
TRANSITION FROM Step1 TO Init
    := xGlobalReset;
END_TRANSITION
STEP Step2:
    xCmmoHomed(S0);
END_STEP
TRANSITION FROM Step2 TO Init
    := Step2.t > T#50ms;
END_TRANSITION
TRANSITION FROM Step2 TO Step4
    := xGlobalReset;
END_TRANSITION
STEP Step4:
    xCmmoHomed(R0);
END_STEP
TRANSITION FROM Step4 TO INIT
    := NOT xCMMOHomed;
END_TRANSITION

END_PROGRAM

// Device/Application/PRGS/prg_DriveZAxis
PROGRAM prg_DriveZAxis
VAR
	uiStep: UINT;
	
END_VAR


CASE uiStep OF
0:	
IF xStartDriveZ THEN
	uiStep := 5;
END_IF


5:
IF uiPositionZToDrive = 1 THEN
	uiStep := 10;	
ELSIF uiPositionZToDrive = 2 THEN
	uiStep := 20;
ELSIF uiPositionZToDrive = 3 THEN
	uiStep := 30;
END_IF

10:
cmmoSTRecord := CMMOSTRecordGrab;
CMMO_WRITE_RECORD_1.usiRecordNo := 3;
CMMO_WRITE_RECORD_1.xExecute := TRUE;
CMMO_MOVE_TO_RECORD_1.usiRecordNo := 1;
uiStep := 40;

20:
cmmoSTRecord := CMMOSTRecordFront;
CMMO_WRITE_RECORD_1.usiRecordNo := 2;
CMMO_WRITE_RECORD_1.xExecute := TRUE;
CMMO_MOVE_TO_RECORD_1.usiRecordNo := 2;
uiStep := 40;

30:
cmmoSTRecord := CMMOSTRecordRear;
CMMO_WRITE_RECORD_1.usiRecordNo := 3;
CMMO_WRITE_RECORD_1.xExecute := TRUE;
CMMO_MOVE_TO_RECORD_1.usiRecordNo := 3;
uiStep := 40;

40:
CMMO_WRITE_RECORD_1.xExecute := FALSE;
IF CMMO_WRITE_RECORD_1.xDONE AND NOT CMMO_WRITE_RECORD_1.xBusy THEN
	uiStep  := 45;
END_IF

45: 
CMMO_MOVE_TO_RECORD_1.xExecute := TRUE;
		IF CMMO_MOVE_TO_RECORD_1.xDone AND NOT CMMO_MOVE_TO_RECORD_1.xBusy THEN
			CMMO_MOVE_TO_RECORD_1.xExecute := FALSE;
			xPositionZReached := TRUE;
			uiStep := 50;
		END_IF
50:

IF xResetZDrive AND NOT xStartDriveZ THEN

	xPositionZReached := FALSE;
	uiStep := 0;
END_IF

END_CASE

END_PROGRAM

// Device/Application/FB/FB_DriveZAxis
FUNCTION_BLOCK FB_DriveZAxis
VAR_INPUT
	uiPosition: UINT; // Positions (1 == GrabPosition; 2 == FrontPosition; 3 == RearPosition)
	xStartDrive: BOOL;
	xReset: BOOL;
END_VAR
VAR_OUTPUT
	xPositionReached: BOOL;
END_VAR
VAR
	uiStep: UINT;
	R_TRIG_Start: R_TRIG;
	TON_Pulse: TON;
END_VAR

//R_TRIG_Start(CLK:= xStartDrive, Q=> );
TON_Pulse(IN:= , PT:= T#100MS, Q=> , ET=> );
CASE uiStep OF
0:	
IF xStartDrive THEN
	uiStep := 5;
END_IF


5:
IF uiPosition = 1 THEN
	uiStep := 10;	
ELSIF uiPosition = 2 THEN
	uiStep := 20;
ELSIF uiPosition = 3 THEN
	uiStep := 30;
END_IF

10:
cmmoSTRecord := CMMOSTRecordGrab;
CMMO_WRITE_RECORD_1.usiRecordNo := 3;
CMMO_WRITE_RECORD_1.xExecute := TRUE;
CMMO_MOVE_TO_RECORD_1.usiRecordNo := 1;
uiStep := 40;

20:
cmmoSTRecord := CMMOSTRecordFront;
CMMO_WRITE_RECORD_1.usiRecordNo := 2;
CMMO_WRITE_RECORD_1.xExecute := TRUE;
CMMO_MOVE_TO_RECORD_1.usiRecordNo := 2;
uiStep := 40;

30:
cmmoSTRecord := CMMOSTRecordRear;
CMMO_WRITE_RECORD_1.usiRecordNo := 3;
CMMO_WRITE_RECORD_1.xExecute := TRUE;
CMMO_MOVE_TO_RECORD_1.usiRecordNo := 3;
uiStep := 40;

40:
CMMO_WRITE_RECORD_1.xExecute := FALSE;
IF CMMO_WRITE_RECORD_1.xDONE AND NOT CMMO_WRITE_RECORD_1.xBusy THEN
	uiStep  := 45;
END_IF

45: 
CMMO_MOVE_TO_RECORD_1.xExecute := TRUE;
		IF CMMO_MOVE_TO_RECORD_1.xDone AND NOT CMMO_MOVE_TO_RECORD_1.xBusy THEN
			CMMO_MOVE_TO_RECORD_1.xExecute := FALSE;
			xPositionReached := TRUE;
			uiStep := 50;
		END_IF
50:
TON_PULSE.IN := TRUE;
IF xReset THEN
	TON_PULSE.IN := FALSE;
	xPositionReached := FALSE;
	uiStep := 0;
END_IF

END_CASE

END_FUNCTION_BLOCK

// Device/Application/FB/FB_Recognize
FUNCTION_BLOCK FB_Recognize
VAR_INPUT
	xReset: BOOL; 	//Reset FB
	xStartRec: BOOL;
END_VAR
VAR_OUTPUT
	bWorkpiece: BYTE; // Erkanntes Werkstück || recognized Workpiece
	xSet: BOOL;
END_VAR
VAR
	uiStep: UINT;
	ixPercLightGate: BOOL;
	// Zählbyte zum erkennen von Transparent
	CountUpLightGate: CTU;
	TON_Set: TON;
	TON_Wait: TON;
	test: WORD;
	TON_WaitForIt: TON;
	RS_Reflex: RS;
	RS_Induct: RS;
END_VAR

CountUpLightGate(
	CU:= , 
	RESET:= xReset, 
	PV:= 2, 
	Q=> , 
	CV=> test);
	
RS_Reflex(SET:= , RESET1:= xReset, Q1=> );
RS_Induct(SET:= , RESET1:= xReset, Q1=> );	
	
	
TON_WaitForIt(IN:= , PT:= T#1S, Q=> , ET=> );
IF xStartRec THEN
	CountUpLightGate.RESET := FALSE;
	IF NOT CountUpLightGate.Q THEN
		CountUpLightGate.CU := ixLightGate;
	END_IF
END_IF

	IF xReset THEN
		bWorkPiece := 99;
		uiStep := 0;
	END_IF
	
CASE uiStep OF
	0:
	xSet := FALSE;
	CountUpLightGate.RESET := FALSE;
	RS_Induct.RESET1 := FALSE;
	RS_Reflex.RESET1 := FALSE;
	IF xStartRec THEN
		uiStep := 2;
	END_IF
	
	2:
	IF ixLightGate THEN
		uiStep := 5;
	END_IF
	
	5:
	TON_WaitForIt.IN := TRUE;
	RS_Reflex.SET := ixPercReflex;
	RS_Induct.SET := ixPercInduct;
	IF TON_WaitForIt.Q THEN
		uiStep := 10;
	END_IF
	
	10:
	TON_WaitForIt.IN := FALSE;
	IF RS_Reflex.Q1 THEN
		bWorkpiece := 0;
	ELSE
		bWorkpiece := 1;
	END_IF
	uiStep := 11;
	
	11:
	IF RS_Induct.Q1 THEN
		bWorkpiece := 2;
	END_IF
	uiStep := 12;
	
(*	IF NOT RS_induct.Q1 AND NOT RS_Reflex.Q1 AND NOT CountUpLightGate.Q THEN
		bWorkpiece := 55;
	END_IF
*)	
	
	12:
	IF CountUpLightGate.Q THEN
		bWorkpiece := 3;
	END_IF
	uiStep := 30;
	
	30:
	xSet := TRUE;
	
	IF xReset THEN
		uiStep := 0;
		bWorkpiece := 0;
		CountUpLightGate.RESET := TRUE;
		RS_Induct.RESET1 := TRUE;
		RS_Reflex.RESET1 := TRUE;
	END_IF
END_CASE

END_FUNCTION_BLOCK

// Device/Application/FB/FB_CalcRackPos
FUNCTION_BLOCK FB_CalcRackPos
VAR_INPUT
	uiShelf:	   	UINT;	
	uiRow: 			UINT;
	rPalettOffset: 	REAL; // Default == 4
	rShelfOffset: 	REAL; // Default == 90

END_VAR
VAR_OUTPUT
	wCalcRackPos_X: WORD;
	wCalcRackPos_Y: WORD;
	
	rCalcRackPos_X: REAL;
	rCalcRackPos_Y: REAL;
END_VAR
VAR

	
	
END_VAR

	rCalcRackPos_X 					:= rXPositionWorkPiece1 - (uiShelf * rShelfOffset);
	rCalcRackPos_Y 					:= rYPositionWorkPiece1 - (uiRow   * rPalettOffset);
	
	wCalcRackPos_X := REAL_TO_WORD((rCalcRackPos_X*10));
	wCalcRackPos_X := REAL_TO_WORD((rCalcRackPos_X*10));

END_FUNCTION_BLOCK

// Device/Application/FB/FB_StoreSearch
FUNCTION_BLOCK FB_StoreSearch
VAR_INPUT
	bRcvData:			 BYTE; // Werkstücktyp  0 == rot, 1 == schwarz, 2 == silber, 3 == transparent .. Wenn xSearchMode = 1 dann entspricht bRcvData dem Regalfach|| Type of Workpiece  0 == red, 1 == black, 2 == silver, 3 == transparent .. If xSearchMode = 0 -> bRcvData == ShelfNumber
	xStart: BOOL;
	xReset: BOOL;
	uiSearchMode: UINT;		 // 0 == AUTO , 1 == REGALFACH//shelf
	uiStoreMode:  UINT;		 // 0 == Einlagern; 1 == Auslagern || 0 == Store ; 1 == Unstore
END_VAR


VAR_OUTPUT
	xStoragePlaceSpotted: 		 BOOL;
	xErrorStorage:				 BOOL;
	uiOutShelfNumber:			 UINT;
	uiOutRow: 					 UINT;
	uiOutRowPlace:				 UINT;
END_VAR
VAR
	uiShelfNumber: 					UINT := 0;
	uiRow:				    		UINT := 0;
	uiRowPlace: 					UINT := 0;
	//uiShelfNumber:				INT := 0;
	i:								UINT := 0;
	uiStep: UINT;

	xDummy: BOOL;
	TON_NoStorePlaceFound: TON;
	TON_ErrorTimer: TON;
END_VAR

TON_NoStorePlaceFound(IN:= , PT:= T#500MS, Q=> , ET=> );

TON_ErrorTimer(IN:= , PT:=T#5S , Q=> , ET=> );

qxStorageFull := FB_StoreSearch1.xErrorStorage;

IF xErrorStorage THEN
	TON_ErrorTimer.IN := TRUE;	
END_IF

IF TON_ErrorTimer.Q THEN			//after 5 seconds Error turns false
	TON_ErrorTimer.IN := FALSE;
	xErrorStorage := FALSE;
END_IF

IF uiStep = 2 THEN
	TON_NoStorePlaceFound.IN := TRUE;
ELSE
	TON_NoStorePlaceFound.IN := FALSE;
END_IF

IF TON_NoStorePlaceFound.Q THEN
	xErrorStorage := TRUE;
END_IF


IF xFail THEN
	xStorePlaceFound := FALSE;
	xStoragePlaceSpotted := FALSE;
END_IF

IF xReset THEN
	bRcvData := 99;
	uiShelfNumber :=0;
	uiRowPlace := 0;
	uiStep :=0;
	xStoragePlaceSpotted := FALSE;
END_IF



CASE uiStep OF
0:	
IF xStart THEN
	

	uiStep := 2;
END_IF

2:
IF uiStoreMode = 0 THEN
	/////////////////////////////////////////////////////////////////////////////////////////////////////////////////////////////////		
	IF uiSearchMode = 0 THEN ///////////////////////////////////// STOREMODE 0 --> SEARCHMODE ///////////////////////////////////////
			
	///////////////////////////////////// SEARCHMODE 0 /////////////////////////////////////// FABRE BEKANNT, Suche Regalfach zum einlagern
	FOR uiShelfNumber := 0 TO 5 DO
			FOR uiRow := 0 TO 3 DO
						FOR uiRowPlace := 0 TO 1 DO	
								
						IF aStore
Place[uiShelfNumber, uiRow, uiRowPlace].xUsed = FALSE THEN		//if the place is empty and the shelf matches the colout StorePlace is found
								IF aUIColorChoose[uiShelfNumber] = bRcvData THEN			//colour and shelf is linked
									xStorePlaceFound := TRUE;
								ELSE
									xStorePlaceFound := FALSE;
								END_IF
						(*	*)		
							IF uiRowPlace = 0 AND aStorePlace[uiShelfNumber, uiRow, 1].kxUsed THEN			//if front is filled and rear is empty, place is inaccesible so Store Place is not found
								xStorePlaceFound := FALSE;	
							END_IF	
						END_IF
						IF xStorePlaceFound THEN
							EXIT;
						END_IF
							// ????????????????????????????????????????
					END_FOR		
	
					IF xStorePlaceFound THEN 
						EXIT;
					END_IF
			END_FOR
			IF xStorePlaceFound THEN 
				EXIT;
			END_IF
	END_FOR
			IF xStorePlaceFound THEN
			uiStep := 5;
			END_IF


	/////////////////////////////////////////////////////////////////////////////////////////////////////////////////////////////////			
	ELSIF uiSearchMode = 1 THEN	
		///////////////////////////////////// SEARCHMODE 1 /////////////////////////////////////// Suche Platz in bestimmten Regalfach zum einlagern
		
		//////////////////////
		CASE bRcvData OF		
			0:
			//uiShelfNumber := aUIColorChoose[0];
			uiShelfNumber := 0;
			1:
			//uiShelfNumber := aUIColorChoose[1];
			uiShelfNumber := 1;
			2:
			//uiShelfNumber := aUIColorChoose[2];
			uiShelfNumber := 2;
			3:
			//uiShelfNumber := aUIColorChoose[3];
			uiShelfNumber := 3;
			4:
			//uiShelfNumber := aUIColorChoose[4];
			uiShelfNumber := 4;
			5:
			//uiShelfNumber := aUIColorChoose[5];	
			uiShelfNumber := 5;		
			END_CASE
		FOR uiRow := 0 TO 3 DO
			
				FOR uiRowPlace := 0 TO 1 DO
					
					IF aStorePlace[uiShelfNumber, uiRow, uiRowPlace].xUsed = FALSE THEN
					xStorePlaceFound := TRUE;
					END_IF
						
					IF uiRowPlace = 0 AND aStorePlace[uiShelfNumber, uiRow, 1].xUsed THEN
					xStorePlaceFound := FALSE;	
					END_IF
					
					IF xStorePlaceFound THEN
						EXIT;
					END_IF
				END_FOR
				IF xStorePlaceFound THEN 
					EXIT;
				END_IF
		
			IF xStorePlaceFound THEN 
					EXIT;
			END_IF
		END_FOR
			
		IF xStorePlaceFound THEN
		uiStep := 5;
		END_IF

		
		
		
		///////////
	END_IF ///////////ENDE SEARCHMODE 1 ///////////
	

ELSIF uiStoreMode = 1 THEN	

	IF uiSearchMode = 0 THEN ///////////////////////////////////// STOREMODE 1 --> SEARCHMODE 0///////////////////////////////////////
		///////////////////////////////////// SEARCHMODE 0 ///////////////////////////////////////  Suche eingegebene Farbe zum auslagern
		FOR uiShelfNumber := 0 TO 5 DO
				FOR uiRow := 0 TO 3 DO
					FOR uiRowPlace := 0 TO 1 DO	
	
						IF aStorePlace[uiShelfNumber, uiRow, uiRowPlace].xUsed = TRUE THEN
								IF aUIColorChoose[uiShelfNumber] = bRcvData THEN
								//	xStorePlaceFound := TRUE; 
				//				ELSE
					//				xStorePlaceFound := FALSE;
							//	END_IF
									
								IF uiRowPlace = 0 AND aStorePlace[uiShelfNumber, uiRow, 1].xUsed THEN
									uiRowPlace := 1;
									xStorePlaceFound := TRUE;
								ELSE
									uiRowPlace := 0;
									xStorePlaceFound := TRUE;	
								END_IF
								END_IF
						END_IF	
						IF xStorePlaceFound THEN
							EXIT;
						END_IF
					
					END_FOR		
	
					IF xStorePlaceFound THEN 
						EXIT;
					END_IF
				END_FOR
			IF xStorePlaceFound THEN 
				EXIT;
			END_IF
		END_FOR 
			IF xStorePlaceFound THEN
			uiStep := 5;
			END_IF
		
	ELSIF uiSearchMode = 1 THEN	 //////////////////////////////////// STOREMODE 1 --> SEARCHMODE 1//////////////////////////////////////
		 ///////////////////////////////////// SEARCHMODE 1 /////////////////////////////////////// Suche in eingegebenen Regalfach zum auslagern
		 
		CASE bRcvData OF								//xSearchMode is False then this is the shelf number
				0:
				//uiShelfNumber := aUIColorChoose[0];
				uiShelfNumber := 0;
				1:
				//uiShelfNumber := aUIColorChoose[1];
				uiShelfNumber := 1;
				2:
				//uiShelfNumber := aUIColorChoose[2];
				uiShelfNumber := 2;
				3:
				//uiShelfNumber := aUIColorChoose[3];
				uiShelfNumber := 3;
				4:
				//uiShelfNumber := aUIColorChoose[4];
				uiShelfNumber := 4;
				5:
				//uiShelfNumber := aUIColorChoose[5];	
				uiShelfNumber := 5;			
		END_CASE
			FOR uiRow := 0 TO 3 DO
				
					FOR uiRowPlace := 0 TO 1 DO
						
						IF aStorePlace[uiShelfNumber, uiRow, uiRowPlace].xUsed = TRUE THEN
						xStorePlaceFound := TRUE;
						END_IF
							
						IF uiRowPlace = 0 AND aStorePlace[uiShelfNumber, uiRow, 1].xUsed THEN
						uiRowPlace := 1;
						xStorePlaceFound := TRUE;	
						END_IF
						
						IF xStorePlaceFound THEN
							EXIT;
						END_IF
					END_FOR
					IF xStorePlaceFound THEN 
						EXIT;
					END_IF
			
				IF xStorePlaceFound THEN 
						EXIT;
				END_IF
			END_FOR
				
			IF xStorePlaceFound THEN
			uiStep := 5;
			END_IF
		 
		 
	END_IF ////////////////////////// ENDE STOREMODE 1, SEARCHMODE 0 //////////////////////////////////
	
END_IF

IF xErrorStorage THEN
	uiStep := 12;;
END_IF

5:

IF uiRowPlace = 0 THEN
	xRowPlaceFront := TRUE;
ELSIF uiRowPlace = 1 THEN
	 xRowPlaceFront := FALSE;
END_IF	
uiOutShelfNumber := uiShelfNumber;
uiOutRow := uiRow;
uiOutRowPlace := uiRowPlace;	
uiStep := 10;

10:

xStoragePlaceSpotted 	:= TRUE;
xStorePlaceFound		:= FALSE;
//evtl. noch reset einbauen
IF xReset THEN
	
uiShelfNumber  			:= 0;
uiRow    				:= 0;
uiRowPlace			 	:= 0;
uiStep := 0;
END_IF

12:
//DUMMYSTEP
IF xReset THEN
	
uiShelfNumber  			:= 0;
uiRow    				:= 0;
uiRowPlace			 	:= 0;
uiStep := 0;
END_IF

END_CASE

END_FUNCTION_BLOCK

// Device/Application/PRGS/prg_startup
PROGRAM prg_startup
VAR
END_VAR

END_PROGRAM

